r1 := WORD_TO_REAL(Rx_IH_MOUT);
pv_IH_KW := r1 / 10; 

is_IH_TIC_al := Rx_IH_AL > 0;
is_IH_TIC_manual := Rx_IH_AM > 0;
ing_IH_TIC_at := Rx_IH_AT_ST <> 0;

r1 := WORD_TO_REAL(Rx_IH_P);
pv_IH_P := r1 / 10; 

r1 := WORD_TO_REAL(Rx_IH_I);
pv_IH_I := r1 / 10; 

r1 := WORD_TO_REAL(Rx_IH_D);
pv_IH_D := r1 / 10;

END_PROGRAM

// ---- POUs/MR_PRG/P13_DI_N_Check.TcPOU
PROGRAM P13_DI_N_Check
VAR	
    T_Rst_off: TON := (PT:=T#1S);
	
	//for ACT_ROT_JOG_INCH();
	t_ROT_INCH: TON;
	pt_ROT_INCH: TIME;
	p_ROT_INCH: R_TRIG;
	p_ROT_JOG_OFF: F_TRIG;
	
	//for Maint
	p_MAINT: R_TRIG;
	p_DO_TEST: R_TRIG;
END_VAR

//for PC Display
BITS1_DI := %IB0;
BITS2_DI := %IB1;
BITS3_DI := %IB2;
BITS4_DI := %IB3;
BITS5_DI := %IB4;
BITS6_DI := %IB5;
BITS7_DI := %IB6;
BITS8_DI := %IB7;
BITS9_DI := %IB8;

//전체 Reset 신호 1초 발생
T_Rst_Off(IN:= cm_RST);
IF T_Rst_Off.Q THEN
	cm_RST := 0; 
END_IF
s_cm_RST := cm_RST;

//Maint Mode Check
p_MAINT(CLK:=(di_MAINT OR cm_MAINT));
IF p_MAINT.Q AND (di_MAINT OR cm_MAINT) AND ing_RCP = 0 AND is_MAKER_login THEN //Maint On
	ing_MAINT := 1; 
END_IF 
IF (di_MAINT = 0 AND cm_MAINT = 0) OR ing_RCP = 1 OR is_MAKER_login = 0 THEN //Maint Off
	ing_MAINT := 0; 
END_IF 

//DO Test Check
p_DO_TEST(CLK:=cm_DO_TEST);	
IF p_DO_TEST.Q AND ing_MAINT THEN
	s_EN_DO_TEST := 1; 
END_IF
IF ing_MAINT = 0 OR cm_DO_TEST = 0 THEN
	s_EN_DO_TEST := 0; 
	cm_DO_TEST := 0;
END_IF
ing_DO_TEST := s_EN_DO_TEST;	

//S01 -N2 Low Check
is_S01_low_al := pv_S01 < N_A_SV_AL[0];
is_S01_low_wn := pv_S01 < N_A_SV_WN[0];

//S02 -H2 Low Check
is_S02_low_al := pv_S02 < N_A_SV_AL[1];
is_S02_low_wn := pv_S02 < N_A_SV_WN[1];

//S03 -NH3 Low Check
is_S03_low_al := pv_S03 < N_A_SV_AL[2];
is_S03_low_wn := pv_S03 < N_A_SV_WN[2];

//S04 -SiH4 Low Check
is_S04_low_al := pv_S04 < N_A_SV_AL[3];
is_S04_low_wn := pv_S04 < N_A_SV_WN[3];

//P01 Reactor Pressure
is_P01_overP_al := pv_P01 > N_A_SV_AL[4];
is_P01_overP_wn := pv_P01 > N_A_SV_WN[4];

//IH Over Temp
is_IH_overT_al := pv_IH > N_A_SV_AL[5];
is_IH_overT_wn := pv_IH > N_A_SV_WN[5];

//Shower Head CW Over Temp
is_SH_CW_overT_al := pv_IH > N_A_SV_AL[6];
is_SH_CW_overT_wn := pv_IH > N_A_SV_WN[6];

//IH Coil CW Over Temp
is_IH_CW_overT_al := pv_IH_CW > N_A_SV_AL[7];
is_IH_CW_overT_wn := pv_IH_CW > N_A_SV_WN[7];

//P03 Exhaust Pressure
is_P03_overP_al := pv_P03 > N_A_SV_AL[8];
is_P03_overP_wn := pv_P03 > N_A_SV_WN[8];

//DOR Pressure
is_DOR_1ATM := pv_S05 >= e_DOR_1ATM;
is_DOR_05ATM := pv_S05 <= e_DOR_05ATM;
is_DOR_01ATM := pv_S05 <= e_DOR_01ATM;

is_SH_opend := di_SH_lo_limit = 0;

//Rotation : Jog & Inching
ACT_ROT_JOG_INCH();

ACTION ACT_ROT_JOG_INCH:

(*

p_ROT_JOG_OFF(CLK:=EN_ROT_JOG);
//jog runable check
EN_ROT_JOG := (di_ROT_Jog OR cm_ROT_JOG) 
				AND EN_ROT_INCH = 0 
				AND (ing_RCP = 0 OR is_ROT_caliOn = 0)  
				AND al_ROT_fail = Off;//jog
//jog speed set				
IF EN_ROT_JOG THEN
	tsv_ROT := s_ROT_JOG_SPD;
	rtm_ROT := 0;
END_IF

IF p_ROT_JOG_OFF.Q THEN
	tsv_ROT := 0;
	rtm_ROT := 0;
END_IF

t_ROT_INCH(PT := pt_ROT_INCH);//inching timer				
//inching runable check				
p_ROT_INCH(CLK := (di_ROT_60 OR cm_ROT_INCH ) AND EN_ROT_JOG = 0 AND (ing_RCP = 0 OR is_ROT_caliOn = 0) );
IF p_ROT_INCH.Q AND do_Rot = 0  THEN
	cm_ROT_INCH := Off;	
	EN_ROT_INCH := On;
END_IF

//inching speed set
IF EN_ROT_INCH THEN
	tsv_ROT := s_ROT_INCH_SPD;
	rtm_ROT := 0;
	pt_ROT_INCH := REAL_TO_TIME(s_ROT_INCH_TM);//inching time set
	t_ROT_INCH.IN := On;
END_IF

//inching end
IF t_ROT_INCH.Q OR al_ROT_fail THEN
	t_ROT_INCH.IN := Off;
	EN_ROT_INCH := Off;
	tsv_ROT := 0;
	rtm_ROT := 0;
END_IF

IF cm_ROT_pulseZero THEN
	cm_ROT_pulseZero := Off;
	pv_ROT_inchPulse := 0;
	pv_ROT_1turnPulse := 0;
END_IF

ing_ROT_jog := EN_ROT_JOG AND do_Rot;
ing_ROT_inch := EN_ROT_INCH AND do_Rot; 

*)
END_ACTION

END_PROGRAM

// ---- POUs/MR_PRG/P15_AI.TcPOU
PROGRAM P15_AI
VAR
	T1: TON := (PT:=T#100MS);
	halfRes: REAL := 16383;//0~5V
	fullRes: REAL := 32767;//0~10V or 4~20mA
	fullRes_KL3152: REAL := 65535;//4~20mA
	dorOffset: REAL := 3276;
	dorResolution: REAL := 13107;
	dorATM: REAL := 760;			
END_VAR


T1(IN:= 1);
IF T1.Q THEN
	T1(IN:= 0);
	//---------------------- ANALOG ---------------------------	
	IF N_MAX[0] > 0 THEN//MFC01 : 0~5V
	 	pv_M01 := N_MAX[0] * XA_M01 / halfRes ;
	 	dev_M01 := (100 * (sv_M01 - pv_M01)) / N_MAX[0];
	END_IF;	
	IF N_MAX[1] > 0 THEN//MFC02 : 0~5V
		pv_M02 := N_MAX[1] * XA_M02 / halfRes ;
	 	dev_M02 := (100 * (sv_M02 - pv_M02)) / N_MAX[1];
	END_IF;	
	IF N_MAX[2] > 0 THEN//MFC03 : 0~5V
		 pv_M03 := N_MAX[2] * XA_M03 / halfRes ;
		 dev_M03 := (100 * (sv_M03 - pv_M03)) / N_MAX[2];
	END_IF;	
	IF N_MAX[3] > 0 THEN//MFC04 : 0~5V
		 pv_M04 := N_MAX[3] * XA_M04 / halfRes ;
		 dev_M04 := (100 * (sv_M04 - pv_M04)) / N_MAX[3];
	END_IF;	
	IF N_MAX[4] > 0 THEN//MFC05 : 0~5V
		 pv_M05 := N_MAX[4] * XA_M05 / halfRes ;
		 dev_M05 := (100 * (sv_M05 - pv_M05)) / N_MAX[4];
	END_IF;	
	IF N_MAX[5] > 0 THEN//MFC06 : 0~5V
		 pv_M06 := N_MAX[5] * XA_M06 / halfRes ;
		 dev_M06 := (100 * (sv_M06 - pv_M06)) / N_MAX[5];
	END_IF;	
	IF N_MAX[6] > 0 THEN//MFC07 : 0~5V
		 pv_M07 := N_MAX[6] * XA_M07 / halfRes ;
		 dev_M07 := (100 * (sv_M07 - pv_M07)) / N_MAX[6];
	END_IF;	
	IF N_MAX[7] > 0 THEN//MFC08 : 0~5V
		 pv_M08 := N_MAX[7] * XA_M08 / halfRes ;
		 dev_M08 := (100 * (sv_M08 - pv_M08)) / N_MAX[7];
	END_IF;	
	IF N_MAX[8] > 0 THEN//MFC09 : 0~5V
		 pv_M09 := N_MAX[8] * XA_M09 / halfRes ;
		 dev_M09 := (100 * (sv_M09 - pv_M09)) / N_MAX[8];
	END_IF;	
	IF N_MAX[9] > 0 THEN//MFC10 : 0~5V
		 pv_M10 := N_MAX[9] * XA_M10 / halfRes ;
		 dev_M10 := (100 * (sv_M10 - pv_M10)) / N_MAX[9];
	END_IF;	
	IF N_MAX[10] > 0 THEN//MFC11 : 0~5V
		 pv_M11 := N_MAX[10] * XA_M11 / halfRes ;
		 dev_M11 := (100 * (sv_M11 - pv_M11)) / N_MAX[10];
	END_IF;	
	IF N_MAX[11] > 0 THEN//MFC12 : 0~5V
		 pv_M12 := N_MAX[11] * XA_M12 / halfRes ;
		 dev_M12 := (100 * (sv_M12 - pv_M12)) / N_MAX[11];
	END_IF;	
	IF N_MAX[12] > 0 THEN//MFC13 : 0~5V
		 pv_M13 := N_MAX[12] * XA_M13 / halfRes ;
		 dev_M13 := (100 * (sv_M13 - pv_M13)) / N_MAX[12];
	END_IF;	
	IF N_MAX[13] > 0 THEN//MFC14 : 0~5V
		 pv_M14 := N_MAX[13] * XA_M14 / halfRes ;
		 dev_M14 := (100 * (sv_M14 - pv_M14)) / N_MAX[13];
	END_IF;	
	IF N_MAX[14] > 0 THEN//MFC15 : 0~5V
		 pv_M15 := N_MAX[14] * XA_M15 / halfRes ;
		 dev_M15 := (100 * (sv_M15 - pv_M15)) / N_MAX[14];
	END_IF;	
	IF N_MAX[15] > 0 THEN//MFC16 : 0~5V
	 	pv_M16 := N_MAX[15] * XA_M16 / halfRes ;
	 	dev_M16 := (100 * (sv_M16 - pv_M16)) / N_MAX[15];
	END_IF;	
	IF N_MAX[16] > 0 THEN//MFC17 : 0~5V
		 pv_M17 := N_MAX[16] * XA_M17 / halfRes ;
		 dev_M17 := (100 * (sv_M17 - pv_M17)) / N_MAX[16];
	END_IF;	
	IF N_MAX[17] > 0 THEN//MFC18 : 0~5V
		 pv_M18 := N_MAX[17] * XA_M18 / halfRes ;
		 dev_M18 := (100 * (sv_M18 - pv_M18)) / N_MAX[17];
	END_IF;	
	IF N_MAX[18] > 0 THEN//MFC19 : 0~5V
		 pv_M19 := N_MAX[18] * XA_M19 / halfRes ;
		 dev_M19 := (100 * (sv_M19 - pv_M19)) / N_MAX[18];
	END_IF;				
	IF N_MAX[19] > 0 THEN//EPC01 : 0~5V
		pv_E01 := N_MAX[19] * XA_E01 / halfRes ;
		dev_E01 := (100 * (sv_E01 - pv_E01)) / N_MAX[19];
	END_IF;	
	IF N_MAX[20] > 0 THEN//EPC02 : 0~5V
		pv_E02 := N_MAX[20] * XA_E02 / halfRes ;
		dev_E02 := (100 * (sv_E02 - pv_E02)) / N_MAX[20];
	END_IF;	
	IF N_MAX[21] > 0 THEN//EPC03 : 0~5V
		pv_E03 := N_MAX[21] * XA_E03 / halfRes ;
		dev_E03 := (100 * (sv_E03 - pv_E03)) / N_MAX[21];
	END_IF;	
	IF N_MAX[22] > 0 THEN//EPC04 : 0~5V
		pv_E04 := N_MAX[22] * XA_E04 / halfRes ;
		dev_E04 := (100 * (sv_E04 - pv_E04)) / N_MAX[22];
	END_IF;	
	IF N_MAX[23] > 0 THEN //EPC05 : 0~5V
		pv_E05 := N_MAX[23] * XA_E05 / halfRes ;
		dev_E05 := (100 * (sv_E05 - pv_E05)) / N_MAX[23];
	END_IF;	
	IF N_MAX[24] > 0 THEN //EPC06 : 0~5V
		pv_E06 := N_MAX[24] * XA_E06 / halfRes ;
		dev_E06 := (100 * (sv_E06 - pv_E06)) / N_MAX[24];
	END_IF;
	IF N_MAX[25] > 0 THEN//EPC07 : 0~5V
		pv_E07 := N_MAX[25] * XA_E07 / halfRes ;
		dev_E07 := (100 * (sv_E07 - pv_E07)) / N_MAX[25];
	END_IF;			
	IF N_MAX[26] > 0 THEN//IH Temp - E3508 
		//pv_IHT := DeviceNet
		dev_IH := (100 * (sv_IH - pv_IH)) / N_MAX[26];
	END_IF;	
	IF N_MAX[27] > 0 THEN//Rotation RPM : 4~20mA      
	   	 pv_Rot := N_MAX[27] * XA_ROT / fullRes_KL3152;
		 dev_ROT := (100 * (sv_ROT - pv_ROT)) / N_MAX[27];
	END_IF;	
	IF N_MAX[28] > 0 THEN//T/V Position(1~100%) : DeviceNet
		//pv_TV := DeviceNet
		dev_POS := (100 * (sv_POS - pv_POS)) / N_MAX[28];
	END_IF;
	IF N_MAX[29] > 0 THEN//T/V Pressure(1~1000 Torr) : DeviceNet
		//pv_P01 := DeviceNet
		dev_P01 := (100 * (sv_P01 - pv_P01)) / N_MAX[29];
	END_IF;	
	IF N_MAX[30] > 0 THEN//Reactor Pressure(10 Torr) : 0~10V
		pv_P02 := N_MAX[30] * XA_P02 / fullRes;
	END_IF;	
	IF N_MAX[31] > 0 THEN//Exhaust Pressure(1000 Torr) : 0~10V   
	   	 pv_P03 := N_MAX[31] * XA_P03 / fullRes;
	END_IF;		
	IF N_MAX[52] > 0 THEN//N2 Pressure : 4~20mA      
		 pv_S01 := N_MAX[52] * XA_S01 / fullRes;
	END_IF;	
	IF N_MAX[53] > 0 THEN//H2 Pressure : 4~20mA      
		 pv_S02 := N_MAX[53] * XA_S02 / fullRes;
	END_IF;	
	IF N_MAX[54] > 0 THEN//NH3 Pressure : 4~20mA       
		 pv_S03 := N_MAX[54] * XA_S03 / fullRes;
	END_IF;	 
	IF N_MAX[55] > 0 THEN//SiH4 Pressure : 4~20mA      
		 pv_S04 := N_MAX[55] * XA_S04 / fullRes;
	END_IF;	
	IF N_MAX[56] > 0 THEN//DOR Pressure : 1~5V      
		 pv_S05 :=  dorATM - (N_MAX[56] * (XA_S05 - dorOffset) / dorResolution);
	END_IF;
				
	//pv_LHT1 := XA_LHT1 * 0.1 ;
	//pv_LHT2 := XA_LHT2 * 0.1 ;
	//pv_LHT3 := XA_LHT3 * 0.1 ;
	//pv_LHT4 := XA_LHT4 * 0.1 ;
	//pv_LHT5 := XA_LHT5 * 0.1 ;
	//pv_LHT6 := XA_LHT6 * 0.1 ;
	//pv_LHT7 := XA_LHT7 * 0.1 ;
	//pv_LHT8 := XA_LHT8 * 0.1 ;
		
	//Shower Head Temp.
	pv_SH_CW  := XA_SH_CW * 0.1 ;	
	//Induction Coil Water Temp
	pv_IH_CW := XA_IH_CW * 0.1 ;
		
    //Induction KW

END_IF;

END_PROGRAM

// ---- POUs/MR_PRG/P21_AL_WN.TcPOU
PROGRAM P21_AL_WN
VAR
	//Analog Deviation Check
	Dev00, Dev01, Dev02, Dev03, Dev04, Dev05, Dev06, Dev07, Dev08, Dev09: FB_DeviationCheck;
	Dev10, Dev11, Dev12, Dev13, Dev14, Dev15, Dev16, Dev17, Dev18, Dev19: FB_DeviationCheck;
	Dev20, Dev21, Dev22, Dev23, Dev24, Dev25, Dev26, Dev27, Dev28, Dev29: FB_DeviationCheck;
		
	//Digital Noise Check
	wNoiseCheckTime: WORD := 100;	
	FB_AL32, FB_AL33, FB_AL34, FB_AL35, FB_AL36, FB_AL37, FB_AL38, FB_AL39: FB_NoiseCheck;	 
	FB_AL40, FB_AL41, FB_AL42, FB_AL43, FB_AL44, FB_AL45, FB_AL46, FB_AL47: FB_NoiseCheck;
	FB_AL48, FB_AL49, FB_AL50, FB_AL51, FB_AL52, FB_AL53, FB_AL54, FB_AL55: FB_NoiseCheck; 
	FB_AL56, FB_AL57, FB_AL58, FB_AL59, FB_AL60, FB_AL61, FB_AL62, FB_AL63: FB_NoiseCheck; 
	FB_AL64, FB_AL65, FB_AL66, FB_AL67, FB_AL68, FB_AL69, FB_AL70, FB_AL71: FB_NoiseCheck; 
	FB_AL72, FB_AL73, FB_AL74, FB_AL75, FB_AL76, FB_AL77, FB_AL78, FB_AL79: FB_NoiseCheck; 
	FB_AL80, FB_AL81, FB_AL82, FB_AL83, FB_AL84, FB_AL85, FB_AL86, FB_AL87: FB_NoiseCheck;
	FB_AL88, FB_AL89, FB_AL90, FB_AL91, FB_AL92, FB_AL93, FB_AL94, FB_AL95: FB_NoiseCheck; 
	FB_AL96, FB_AL97, FB_AL98, FB_AL99, FB_AL100, FB_AL101, FB_AL102, FB_AL103: FB_NoiseCheck; 
	FB_AL104, FB_AL105, FB_AL106, FB_AL107, FB_AL108, FB_AL109, FB_AL110, FB_AL111: FB_NoiseCheck;
	//FB_AL112, FB_AL113, FB_AL114, FB_AL115, FB_AL116, FB_AL117, FB_AL118, FB_AL119: FB_NoiseCheck; 
	FB_AL120, FB_AL121, FB_AL122, FB_AL123, FB_AL124, FB_AL125, FB_AL126, FB_AL127: FB_NoiseCheck;
	FB_AL128, FB_AL129, FB_AL130, FB_AL131, FB_AL132, FB_AL133, FB_AL134, FB_AL135: FB_NoiseCheck;
	FB_AL136, FB_AL137, FB_AL138, FB_AL139, FB_AL140, FB_AL141, FB_AL142, FB_AL143: FB_NoiseCheck;
	//FB_AL144, FB_AL145, FB_AL146, FB_AL147, FB_AL148, FB_AL149, FB_AL150, FB_AL151: FB_NoiseCheck;
	//FB_AL152, FB_AL153, FB_AL154, FB_AL155, FB_AL156, FB_AL157, FB_AL158, FB_AL159: FB_NoiseCheck;	
			
	FB_WN32, FB_WN33, FB_WN34, FB_WN35, FB_WN36, FB_WN37, FB_WN38, FB_WN39: FB_NoiseCheck; 
	FB_WN40, FB_WN41, FB_WN42, FB_WN43, FB_WN44, FB_WN45, FB_WN46, FB_WN47, FB_WN48, FB_WN49: FB_NoiseCheck; 
	FB_WN50, FB_WN51, FB_WN52, FB_WN53, FB_WN54, FB_WN55, FB_WN56, FB_WN57, FB_WN58, FB_WN59: FB_NoiseCheck; 
	FB_WN60, FB_WN61, FB_WN62, FB_WN63: FB_NoiseCheck;
									
	i: INT;
	bReset: BOOL;
	P_AL_Trig: R_TRIG;
	P_WN_Trig: R_TRIG;
	
	P_di_RST: R_TRIG;
		
	//Real Address
	n_AL_WORD AT%MB38: ARRAY[0..8] OF WORD; //16Bit
	n_WN_DWORD AT%MB56: ARRAY[0..1] OF DWORD; //32Bit
		
	n_AL_WORD_OLD: ARRAY[0..8] OF DWORD; //128EA
	n_WN_DWORD_OLD: ARRAY[0..1] OF DWORD; //64EA
	
	T1S_WN: TON;
	n_BZ_Order: ARRAY[0..1] OF BYTE;//부저 울림 순서, 1 -> Warning, 2 -> Alarm, 1 + 2 = 3 -> Alarm

END_VAR

A_AL_WN_Check();
D_AL_Check();
D_WN_Check();

is_AL := n_AL_WORD[0] > 0 OR n_AL_WORD[1] > 0 OR n_AL_WORD[2] > 0 OR n_AL_WORD[3] > 0 OR n_AL_WORD[4] > 0 OR
		 n_AL_WORD[5] > 0 OR n_AL_WORD[6] > 0 OR n_AL_WORD[7] > 0 OR n_AL_WORD[8] > 0;

is_WN := n_WN_DWORD[0] > 0 OR n_WN_DWORD[1] > 0 ;

//Alarm Processing
D_AL_Check();

//Alarm & Warning Reset
bReset := s_cm_RST;
 IF bReset THEN
	 s_is_DOR_Broken := 0;
 END_IF

//New AL Check
P_AL_Trig(CLK:= n_AL_WORD[0] > n_AL_WORD_OLD[0] OR n_AL_WORD[1] > n_AL_WORD_OLD[1] OR 
			  n_AL_WORD[2] > n_AL_WORD_OLD[2] OR n_AL_WORD[3] > n_AL_WORD_OLD[3] OR
			  n_AL_WORD[4] > n_AL_WORD_OLD[4] OR n_AL_WORD[5] > n_AL_WORD_OLD[5] OR
			  n_AL_WORD[6] > n_AL_WORD_OLD[6] OR n_AL_WORD[7] > n_AL_WORD_OLD[7] OR
			  n_AL_WORD[8] > n_AL_WORD_OLD[8]);
//New WN Check	
P_WN_Trig(CLK:= n_WN_DWORD[0] > n_WN_DWORD_OLD[0] OR n_WN_DWORD[1] > n_WN_DWORD_OLD[1]);

P_di_RST(CLK:= di_RST);	

//AL Backup	
FOR i := 0 TO 8 DO
	n_AL_WORD_OLD[i] := n_AL_WORD[i];
END_FOR
//WN Backup
FOR i := 0 TO 1 DO
	n_WN_DWORD_OLD[i] := n_WN_DWORD[i];
END_FOR

ACTION A_AL_WN_Check:
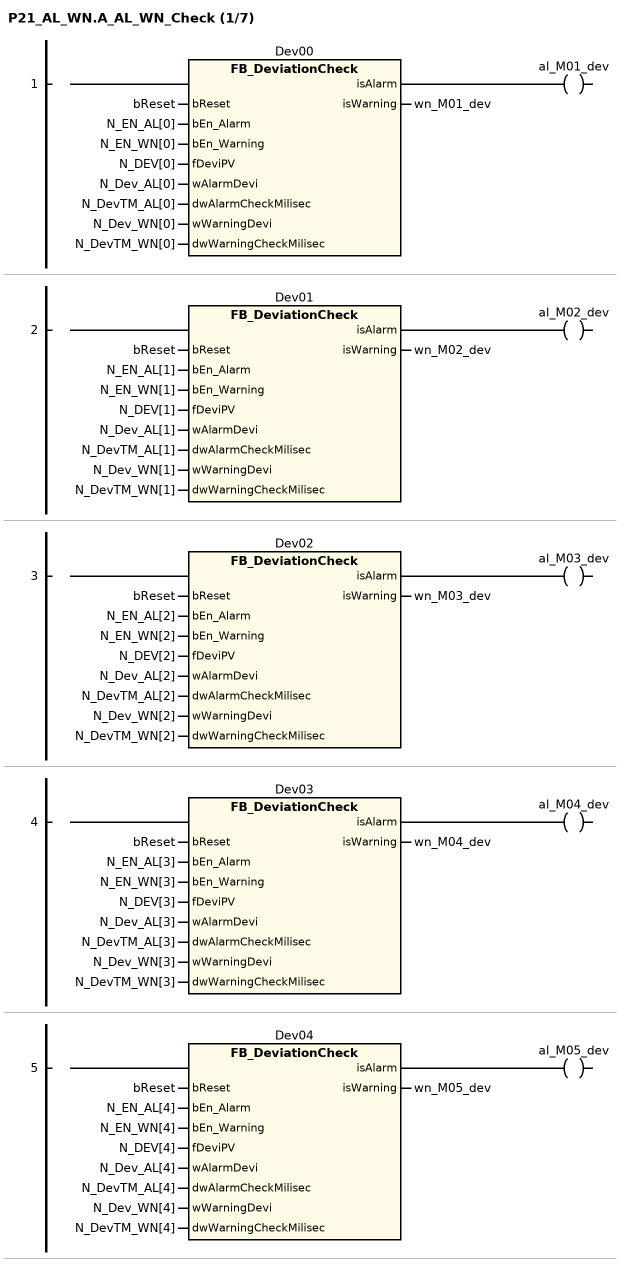
// NETWORK 1
Dev00(
    bReset := bReset,
    bEn_Alarm := N_EN_AL[0],
    bEn_Warning := N_EN_WN[0],
    fDeviPV := N_DEV[0],
    wAlarmDevi := N_Dev_AL[0],
    dwAlarmCheckMilisec := N_DevTM_AL[0],
    wWarningDevi := N_Dev_WN[0],
    dwWarningCheckMilisec := N_DevTM_WN[0],
    isWarning => wn_M01_dev); // FB_DeviationCheck
al_M01_dev := Dev00.isAlarm;

// NETWORK 2
Dev01(
    bReset := bReset,
    bEn_Alarm := N_EN_AL[1],
    bEn_Warning := N_EN_WN[1],
    fDeviPV := N_DEV[1],
    wAlarmDevi := N_Dev_AL[1],
    dwAlarmCheckMilisec := N_DevTM_AL[1],
    wWarningDevi := N_Dev_WN[1],
    dwWarningCheckMilisec := N_DevTM_WN[1],
    isWarning => wn_M02_dev); // FB_DeviationCheck
al_M02_dev := Dev01.isAlarm;

// NETWORK 3
Dev02(
    bReset := bReset,
    bEn_Alarm := N_EN_AL[2],
    bEn_Warning := N_EN_WN[2],
    fDeviPV := N_DEV[2],
    wAlarmDevi := N_Dev_AL[2],
    dwAlarmCheckMilisec := N_DevTM_AL[2],
    wWarningDevi := N_Dev_WN[2],
    dwWarningCheckMilisec := N_DevTM_WN[2],
    isWarning => wn_M03_dev); // FB_DeviationCheck
al_M03_dev := Dev02.isAlarm;

// NETWORK 4
Dev03(
    bReset := bReset,
    bEn_Alarm := N_EN_AL[3],
    bEn_Warning := N_EN_WN[3],
    fDeviPV := N_DEV[3],
    wAlarmDevi := N_Dev_AL[3],
    dwAlarmCheckMilisec := N_DevTM_AL[3],
    wWarningDevi := N_Dev_WN[3],
    dwWarningCheckMilisec := N_DevTM_WN[3],
    isWarning => wn_M04_dev); // FB_DeviationCheck
al_M04_dev := Dev03.isAlarm;

// NETWORK 5
Dev04(
    bReset := bReset,
    bEn_Alarm := N_EN_AL[4],
    bEn_Warning := N_EN_WN[4],
    fDeviPV := N_DEV[4],
    wAlarmDevi := N_Dev_AL[4],
    dwAlarmCheckMilisec := N_DevTM_AL[4],
    wWarningDevi := N_Dev_WN[4],
    dwWarningCheckMilisec := N_DevTM_WN[4],
    isWarning => wn_M05_dev); // FB_DeviationCheck
al_M05_dev := Dev04.isAlarm;

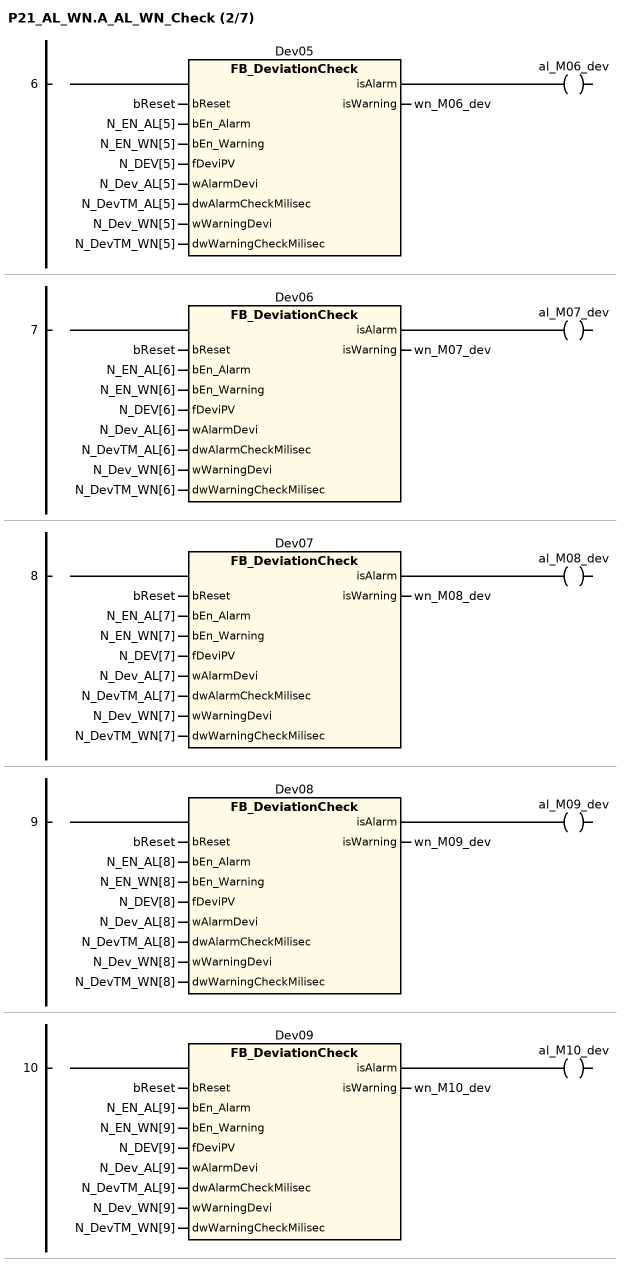
// NETWORK 6
Dev05(
    bReset := bReset,
    bEn_Alarm := N_EN_AL[5],
    bEn_Warning := N_EN_WN[5],
    fDeviPV := N_DEV[5],
    wAlarmDevi := N_Dev_AL[5],
    dwAlarmCheckMilisec := N_DevTM_AL[5],
    wWarningDevi := N_Dev_WN[5],
    dwWarningCheckMilisec := N_DevTM_WN[5],
    isWarning => wn_M06_dev); // FB_DeviationCheck
al_M06_dev := Dev05.isAlarm;

// NETWORK 7
Dev06(
    bReset := bReset,
    bEn_Alarm := N_EN_AL[6],
    bEn_Warning := N_EN_WN[6],
    fDeviPV := N_DEV[6],
    wAlarmDevi := N_Dev_AL[6],
    dwAlarmCheckMilisec := N_DevTM_AL[6],
    wWarningDevi := N_Dev_WN[6],
    dwWarningCheckMilisec := N_DevTM_WN[6],
    isWarning => wn_M07_dev); // FB_DeviationCheck
al_M07_dev := Dev06.isAlarm;

// NETWORK 8
Dev07(
    bReset := bReset,
    bEn_Alarm := N_EN_AL[7],
    bEn_Warning := N_EN_WN[7],
    fDeviPV := N_DEV[7],
    wAlarmDevi := N_Dev_AL[7],
    dwAlarmCheckMilisec := N_DevTM_AL[7],
    wWarningDevi := N_Dev_WN[7],
    dwWarningCheckMilisec := N_DevTM_WN[7],
    isWarning => wn_M08_dev); // FB_DeviationCheck
al_M08_dev := Dev07.isAlarm;

// NETWORK 9
Dev08(
    bReset := bReset,
    bEn_Alarm := N_EN_AL[8],
    bEn_Warning := N_EN_WN[8],
    fDeviPV := N_DEV[8],
    wAlarmDevi := N_Dev_AL[8],
    dwAlarmCheckMilisec := N_DevTM_AL[8],
    wWarningDevi := N_Dev_WN[8],
    dwWarningCheckMilisec := N_DevTM_WN[8],
    isWarning => wn_M09_dev); // FB_DeviationCheck
al_M09_dev := Dev08.isAlarm;

// NETWORK 10
Dev09(
    bReset := bReset,
    bEn_Alarm := N_EN_AL[9],
    bEn_Warning := N_EN_WN[9],
    fDeviPV := N_DEV[9],
    wAlarmDevi := N_Dev_AL[9],
    dwAlarmCheckMilisec := N_DevTM_AL[9],
    wWarningDevi := N_Dev_WN[9],
    dwWarningCheckMilisec := N_DevTM_WN[9],
    isWarning => wn_M10_dev); // FB_DeviationCheck
al_M10_dev := Dev09.isAlarm;

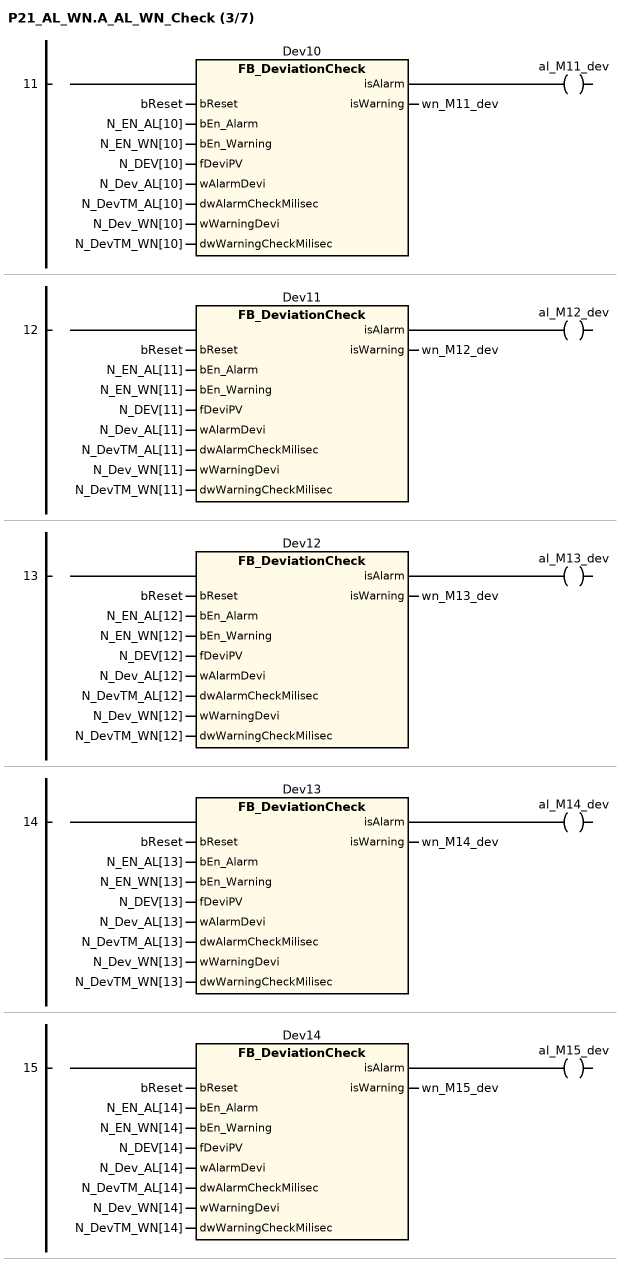
// NETWORK 11
Dev10(
    bReset := bReset,
    bEn_Alarm := N_EN_AL[10],
    bEn_Warning := N_EN_WN[10],
    fDeviPV := N_DEV[10],
    wAlarmDevi := N_Dev_AL[10],
    dwAlarmCheckMilisec := N_DevTM_AL[10],
    wWarningDevi := N_Dev_WN[10],
    dwWarningCheckMilisec := N_DevTM_WN[10],
    isWarning => wn_M11_dev); // FB_DeviationCheck
al_M11_dev := Dev10.isAlarm;

// NETWORK 12
Dev11(
    bReset := bReset,
    bEn_Alarm := N_EN_AL[11],
    bEn_Warning := N_EN_WN[11],
    fDeviPV := N_DEV[11],
    wAlarmDevi := N_Dev_AL[11],
    dwAlarmCheckMilisec := N_DevTM_AL[11],
    wWarningDevi := N_Dev_WN[11],
    dwWarningCheckMilisec := N_DevTM_WN[11],
    isWarning => wn_M12_dev); // FB_DeviationCheck
al_M12_dev := Dev11.isAlarm;

// NETWORK 13
Dev12(
    bReset := bReset,
    bEn_Alarm := N_EN_AL[12],
    bEn_Warning := N_EN_WN[12],
    fDeviPV := N_DEV[12],
    wAlarmDevi := N_Dev_AL[12],
    dwAlarmCheckMilisec := N_DevTM_AL[12],
    wWarningDevi := N_Dev_WN[12],
    dwWarningCheckMilisec := N_DevTM_WN[12],
    isWarning => wn_M13_dev); // FB_DeviationCheck
al_M13_dev := Dev12.isAlarm;

// NETWORK 14
Dev13(
    bReset := bReset,
    bEn_Alarm := N_EN_AL[13],
    bEn_Warning := N_EN_WN[13],
    fDeviPV := N_DEV[13],
    wAlarmDevi := N_Dev_AL[13],
    dwAlarmCheckMilisec := N_DevTM_AL[13],
    wWarningDevi := N_Dev_WN[13],
    dwWarningCheckMilisec := N_DevTM_WN[13],
    isWarning => wn_M14_dev); // FB_DeviationCheck
al_M14_dev := Dev13.isAlarm;

// NETWORK 15
Dev14(
    bReset := bReset,
    bEn_Alarm := N_EN_AL[14],
    bEn_Warning := N_EN_WN[14],
    fDeviPV := N_DEV[14],
    wAlarmDevi := N_Dev_AL[14],
    dwAlarmCheckMilisec := N_DevTM_AL[14],
    wWarningDevi := N_Dev_WN[14],
    dwWarningCheckMilisec := N_DevTM_WN[14],
    isWarning => wn_M15_dev); // FB_DeviationCheck
al_M15_dev := Dev14.isAlarm;

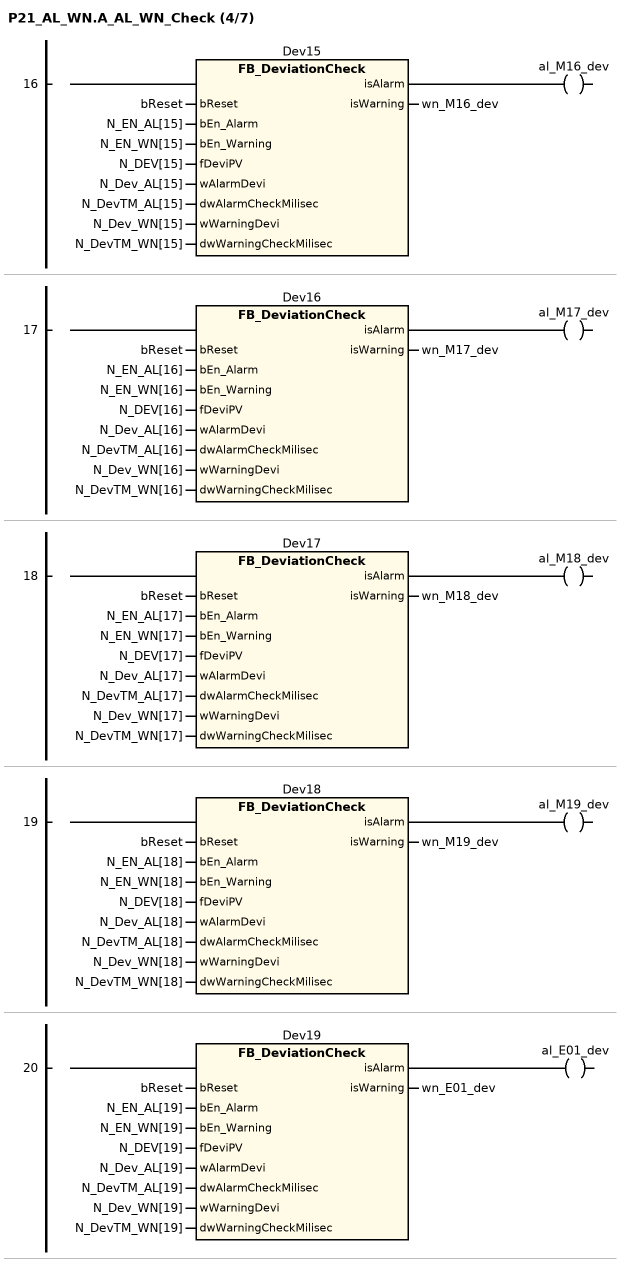
// NETWORK 16
Dev15(
    bReset := bReset,
    bEn_Alarm := N_EN_AL[15],
    bEn_Warning := N_EN_WN[15],
    fDeviPV := N_DEV[15],
    wAlarmDevi := N_Dev_AL[15],
    dwAlarmCheckMilisec := N_DevTM_AL[15],
    wWarningDevi := N_Dev_WN[15],
    dwWarningCheckMilisec := N_DevTM_WN[15],
    isWarning => wn_M16_dev); // FB_DeviationCheck
al_M16_dev := Dev15.isAlarm;

// NETWORK 17
Dev16(
    bReset := bReset,
    bEn_Alarm := N_EN_AL[16],
    bEn_Warning := N_EN_WN[16],
    fDeviPV := N_DEV[16],
    wAlarmDevi := N_Dev_AL[16],
    dwAlarmCheckMilisec := N_DevTM_AL[16],
    wWarningDevi := N_Dev_WN[16],
    dwWarningCheckMilisec := N_DevTM_WN[16],
    isWarning => wn_M17_dev); // FB_DeviationCheck
al_M17_dev := Dev16.isAlarm;

// NETWORK 18
Dev17(
    bReset := bReset,
    bEn_Alarm := N_EN_AL[17],
    bEn_Warning := N_EN_WN[17],
    fDeviPV := N_DEV[17],
    wAlarmDevi := N_Dev_AL[17],
    dwAlarmCheckMilisec := N_DevTM_AL[17],
    wWarningDevi := N_Dev_WN[17],
    dwWarningCheckMilisec := N_DevTM_WN[17],
    isWarning => wn_M18_dev); // FB_DeviationCheck
al_M18_dev := Dev17.isAlarm;

// NETWORK 19
Dev18(
    bReset := bReset,
    bEn_Alarm := N_EN_AL[18],
    bEn_Warning := N_EN_WN[18],
    fDeviPV := N_DEV[18],
    wAlarmDevi := N_Dev_AL[18],
    dwAlarmCheckMilisec := N_DevTM_AL[18],
    wWarningDevi := N_Dev_WN[18],
    dwWarningCheckMilisec := N_DevTM_WN[18],
    isWarning => wn_M19_dev); // FB_DeviationCheck
al_M19_dev := Dev18.isAlarm;

// NETWORK 20
Dev19(
    bReset := bReset,
    bEn_Alarm := N_EN_AL[19],
    bEn_Warning := N_EN_WN[19],
    fDeviPV := N_DEV[19],
    wAlarmDevi := N_Dev_AL[19],
    dwAlarmCheckMilisec := N_DevTM_AL[19],
    wWarningDevi := N_Dev_WN[19],
    dwWarningCheckMilisec := N_DevTM_WN[19],
    isWarning => wn_E01_dev); // FB_DeviationCheck
al_E01_dev := Dev19.isAlarm;

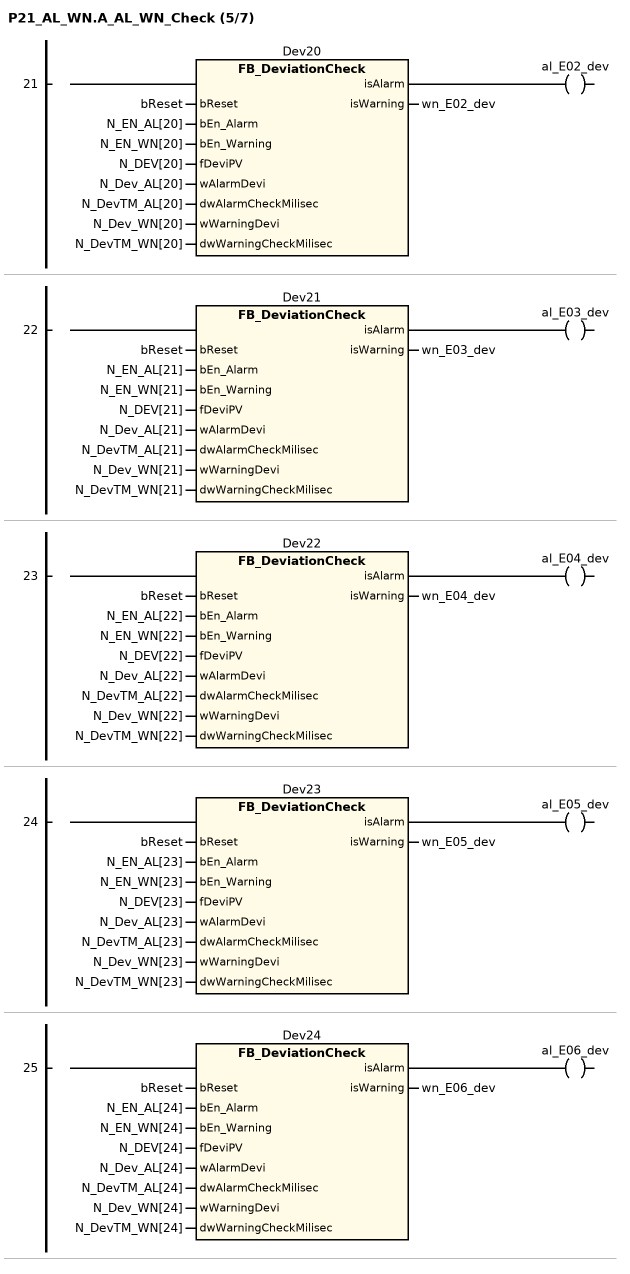
// NETWORK 21
Dev20(
    bReset := bReset,
    bEn_Alarm := N_EN_AL[20],
    bEn_Warning := N_EN_WN[20],
    fDeviPV := N_DEV[20],
    wAlarmDevi := N_Dev_AL[20],
    dwAlarmCheckMilisec := N_DevTM_AL[20],
    wWarningDevi := N_Dev_WN[20],
    dwWarningCheckMilisec := N_DevTM_WN[20],
    isWarning => wn_E02_dev); // FB_DeviationCheck
al_E02_dev := Dev20.isAlarm;

// NETWORK 22
Dev21(
    bReset := bReset,
    bEn_Alarm := N_EN_AL[21],
    bEn_Warning := N_EN_WN[21],
    fDeviPV := N_DEV[21],
    wAlarmDevi := N_Dev_AL[21],
    dwAlarmCheckMilisec := N_DevTM_AL[21],
    wWarningDevi := N_Dev_WN[21],
    dwWarningCheckMilisec := N_DevTM_WN[21],
    isWarning => wn_E03_dev); // FB_DeviationCheck
al_E03_dev := Dev21.isAlarm;

// NETWORK 23
Dev22(
    bReset := bReset,
    bEn_Alarm := N_EN_AL[22],
    bEn_Warning := N_EN_WN[22],
    fDeviPV := N_DEV[22],
    wAlarmDevi := N_Dev_AL[22],
    dwAlarmCheckMilisec := N_DevTM_AL[22],
    wWarningDevi := N_Dev_WN[22],
    dwWarningCheckMilisec := N_DevTM_WN[22],
    isWarning => wn_E04_dev); // FB_DeviationCheck
al_E04_dev := Dev22.isAlarm;

// NETWORK 24
Dev23(
    bReset := bReset,
    bEn_Alarm := N_EN_AL[23],
    bEn_Warning := N_EN_WN[23],
    fDeviPV := N_DEV[23],
    wAlarmDevi := N_Dev_AL[23],
    dwAlarmCheckMilisec := N_DevTM_AL[23],
    wWarningDevi := N_Dev_WN[23],
    dwWarningCheckMilisec := N_DevTM_WN[23],
    isWarning => wn_E05_dev); // FB_DeviationCheck
al_E05_dev := Dev23.isAlarm;

// NETWORK 25
Dev24(
    bReset := bReset,
    bEn_Alarm := N_EN_AL[24],
    bEn_Warning := N_EN_WN[24],
    fDeviPV := N_DEV[24],
    wAlarmDevi := N_Dev_AL[24],
    dwAlarmCheckMilisec := N_DevTM_AL[24],
    wWarningDevi := N_Dev_WN[24],
    dwWarningCheckMilisec := N_DevTM_WN[24],
    isWarning => wn_E06_dev); // FB_DeviationCheck
al_E06_dev := Dev24.isAlarm;

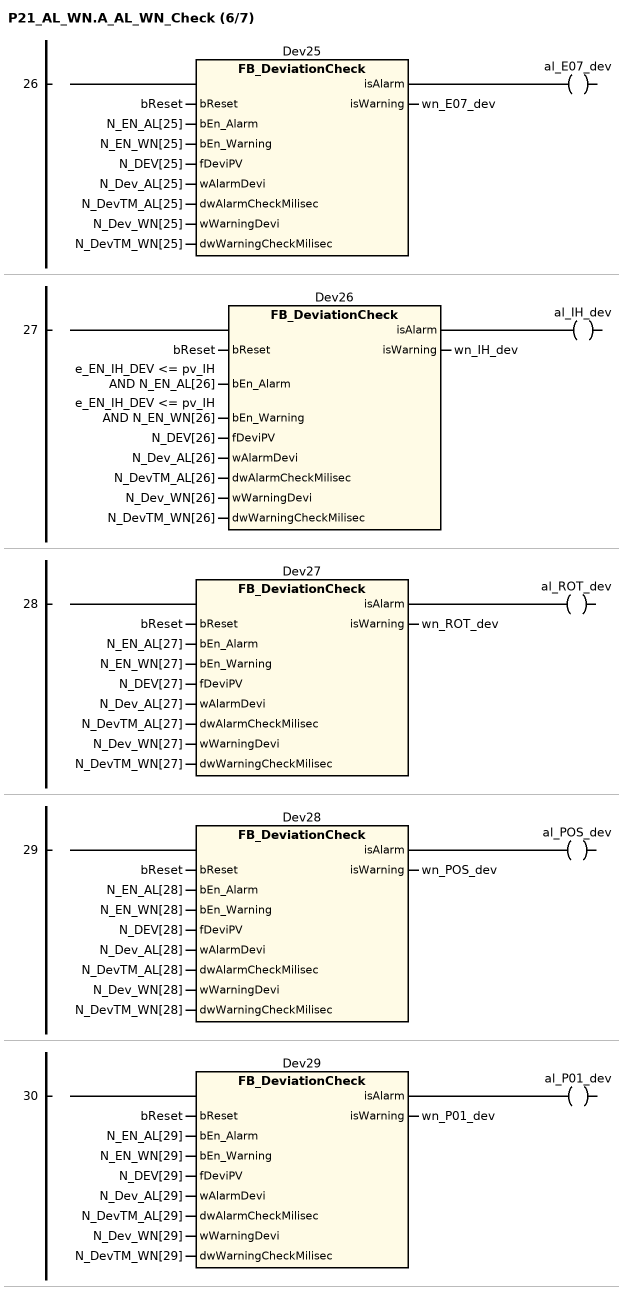
// NETWORK 26
Dev25(
    bReset := bReset,
    bEn_Alarm := N_EN_AL[25],
    bEn_Warning := N_EN_WN[25],
    fDeviPV := N_DEV[25],
    wAlarmDevi := N_Dev_AL[25],
    dwAlarmCheckMilisec := N_DevTM_AL[25],
    wWarningDevi := N_Dev_WN[25],
    dwWarningCheckMilisec := N_DevTM_WN[25],
    isWarning => wn_E07_dev); // FB_DeviationCheck
al_E07_dev := Dev25.isAlarm;

// NETWORK 27
Dev26(
    bReset := bReset,
    bEn_Alarm := e_EN_IH_DEV <= pv_IH AND N_EN_AL[26],
    bEn_Warning := e_EN_IH_DEV <= pv_IH AND N_EN_WN[26],
    fDeviPV := N_DEV[26],
    wAlarmDevi := N_Dev_AL[26],
    dwAlarmCheckMilisec := N_DevTM_AL[26],
    wWarningDevi := N_Dev_WN[26],
    dwWarningCheckMilisec := N_DevTM_WN[26],
    isWarning => wn_IH_dev); // FB_DeviationCheck
al_IH_dev := Dev26.isAlarm;

// NETWORK 28
Dev27(
    bReset := bReset,
    bEn_Alarm := N_EN_AL[27],
    bEn_Warning := N_EN_WN[27],
    fDeviPV := N_DEV[27],
    wAlarmDevi := N_Dev_AL[27],
    dwAlarmCheckMilisec := N_DevTM_AL[27],
    wWarningDevi := N_Dev_WN[27],
    dwWarningCheckMilisec := N_DevTM_WN[27],
    isWarning => wn_ROT_dev); // FB_DeviationCheck
al_ROT_dev := Dev27.isAlarm;

// NETWORK 29
Dev28(
    bReset := bReset,
    bEn_Alarm := N_EN_AL[28],
    bEn_Warning := N_EN_WN[28],
    fDeviPV := N_DEV[28],
    wAlarmDevi := N_Dev_AL[28],
    dwAlarmCheckMilisec := N_DevTM_AL[28],
    wWarningDevi := N_Dev_WN[28],
    dwWarningCheckMilisec := N_DevTM_WN[28],
    isWarning => wn_POS_dev); // FB_DeviationCheck
al_POS_dev := Dev28.isAlarm;

// NETWORK 30
Dev29(
    bReset := bReset,
    bEn_Alarm := N_EN_AL[29],
    bEn_Warning := N_EN_WN[29],
    fDeviPV := N_DEV[29],
    wAlarmDevi := N_Dev_AL[29],
    dwAlarmCheckMilisec := N_DevTM_AL[29],
    wWarningDevi := N_Dev_WN[29],
    dwWarningCheckMilisec := N_DevTM_WN[29],
    isWarning => wn_P01_dev); // FB_DeviationCheck
al_P01_dev := Dev29.isAlarm;

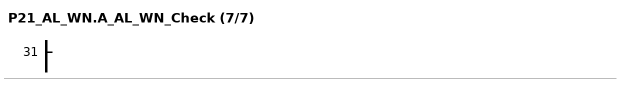
// NETWORK 31
END_ACTION

ACTION Cause_N_Effect:

//WN Buzzer
IF P_WN_Trig.Q THEN
	IF n_BZ_Order[0] <= 0 THEN
		n_BZ_Order[0] := 1; 
	ELSE
		IF n_BZ_Order[0] <> 1 THEN
			n_BZ_Order[1] := 1;
		END_IF
	END_IF
END_IF

//new Alarm rised
IF P_AL_Trig.Q THEN	
	//AL Buzzer
	IF n_BZ_Order[0] <= 0 THEN
		n_BZ_Order[0] := 2; 
	ELSE
		IF n_BZ_Order[0] <> 2 THEN
			n_BZ_Order[1] := 2;
		END_IF
	END_IF
	//AL UserState	
	IF e_US_AL > 0 THEN
		CASE e_US_AL OF
			1: cm_US1 := 1;
			2: cm_US2 := 1;
			3: cm_US3 := 1;
			4: cm_US4 := 1;
		END_CASE
	END_IF	
END_IF	

//IHT 
IF al_PCW_low OR al_IH_fail OR al_IH_overT OR al_SH_CW_overT OR al_IH_CW_overT THEN
	cm_IH := 0;
END_IF
					 
//H2 & SiH4 & NH3
IF is_AL THEN	
	cm_V01 := 0;// H2 Supply
	cm_V02 := 0;// H2 Supply
	cm_V03 := 0;//SiH4 Supply
	cm_V04 := 0;//NH3 Supply
END_IF

IF is_P01_overP_al THEN //둘다 닫아 자연스럽게 동자
	cm_V33_1 := 0;
	cm_V33_2 := 0;
END_IF

IF al_DOR OR wn_DOR THEN
	s_DOR_CNT := 0;
END_IF


//Buzzer Off Process
IF cm_BZ_UserStop OR P_di_RST.Q THEN
	IF n_BZ_Order[0] > 0 THEN
		n_BZ_Order[0] := 0; 
	ELSE
		n_BZ_Order[1] := 0;
	END_IF
	cm_BZ := 0;
	cm_BZ_UserStop := 0; 
END_IF

//Buzzer On Process
IF ing_Maint = 0 THEN	
	T1S_WN(PT:=T#1S);
	T1S_WN.IN :=  n_BZ_Order[0] + n_BZ_Order[1] = 1;
	IF T1S_WN.Q THEN //warning buzzer is 1sec cycle
		T1S_WN.IN := 0;
		cm_BZ := NOT cm_BZ;
	END_IF
	
	IF n_BZ_Order[0] + n_BZ_Order[1] >= 2 THEN
		cm_BZ := 1;
	END_IF
END_IF


//H2	
//IF al_N2_Low OR  al_H2_Low OR al_NH3_Low OR al_GC_H2_Leak OR al_RC_H2_Leak  THEN 
	//H2 Valve OFF - kjk??
	//cm_V27 := OFF;
//END_IF

//EMG_InductionPower
(*IF al_CW_IH_TempHi = ON THEN
	do_IH_Pow := OFF;
ELSE
	IF al_CHM_TempHi = ON THEN
		do_IH_Pow := OFF;
	ELSE
		IF al_GC_H2_Leak = ON THEN
			do_IH_Pow := OFF;
		ELSE
			IF al_RC_H2_Leak = ON THEN
				do_IH_Pow := OFF;
			ELSE
				do_IH_Pow := ON;	
			END_IF		
		END_IF		
	END_IF		
END_IF *)
END_ACTION

ACTION D_AL_Check:
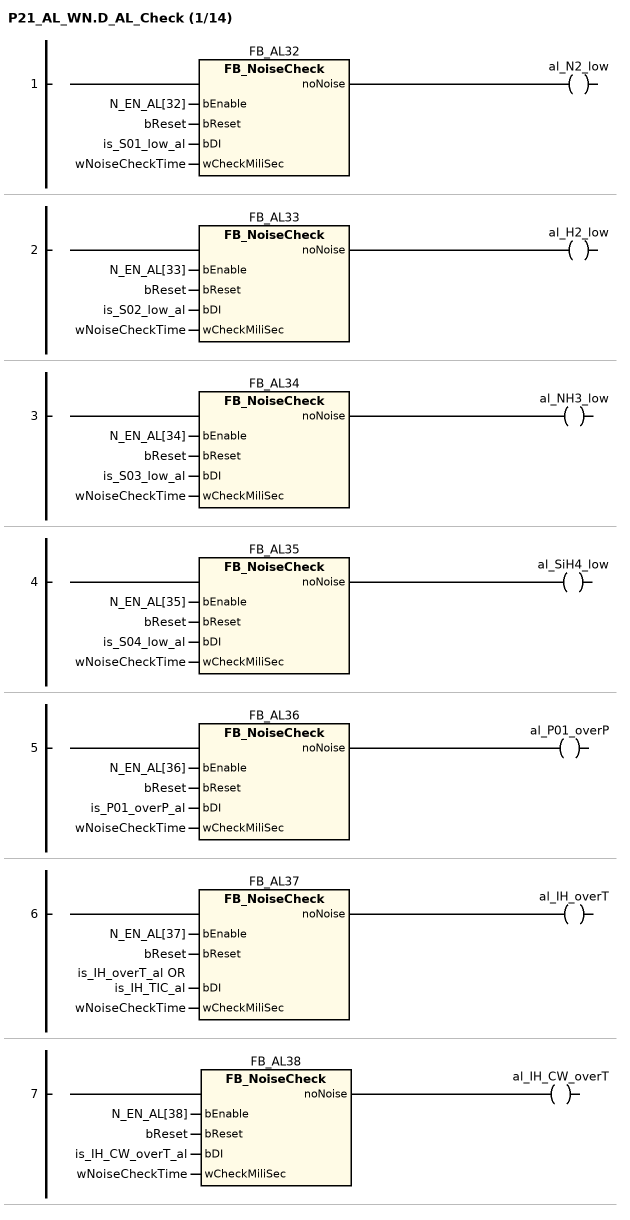
// NETWORK 1
FB_AL32(bEnable := N_EN_AL[32], bReset := bReset, bDI := is_S01_low_al, wCheckMiliSec := wNoiseCheckTime); // FB_NoiseCheck
al_N2_low := FB_AL32.noNoise;

// NETWORK 2
FB_AL33(bEnable := N_EN_AL[33], bReset := bReset, bDI := is_S02_low_al, wCheckMiliSec := wNoiseCheckTime); // FB_NoiseCheck
al_H2_low := FB_AL33.noNoise;

// NETWORK 3
FB_AL34(bEnable := N_EN_AL[34], bReset := bReset, bDI := is_S03_low_al, wCheckMiliSec := wNoiseCheckTime); // FB_NoiseCheck
al_NH3_low := FB_AL34.noNoise;

// NETWORK 4
FB_AL35(bEnable := N_EN_AL[35], bReset := bReset, bDI := is_S04_low_al, wCheckMiliSec := wNoiseCheckTime); // FB_NoiseCheck
al_SiH4_low := FB_AL35.noNoise;

// NETWORK 5
FB_AL36(bEnable := N_EN_AL[36], bReset := bReset, bDI := is_P01_overP_al, wCheckMiliSec := wNoiseCheckTime); // FB_NoiseCheck
al_P01_overP := FB_AL36.noNoise;

// NETWORK 6
FB_AL37(
    bEnable := N_EN_AL[37],
    bReset := bReset,
    bDI := is_IH_overT_al OR is_IH_TIC_al,
    wCheckMiliSec := wNoiseCheckTime); // FB_NoiseCheck
al_IH_overT := FB_AL37.noNoise;

// NETWORK 7
FB_AL38(bEnable := N_EN_AL[38], bReset := bReset, bDI := is_IH_CW_overT_al, wCheckMiliSec := wNoiseCheckTime); // FB_NoiseCheck
al_IH_CW_overT := FB_AL38.noNoise;

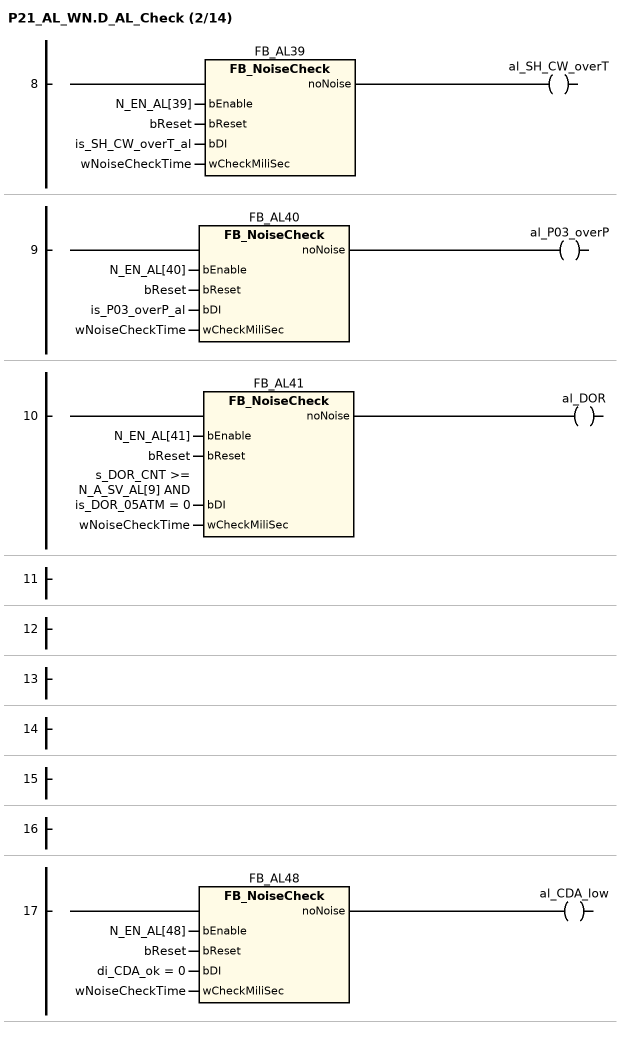
// NETWORK 8
FB_AL39(bEnable := N_EN_AL[39], bReset := bReset, bDI := is_SH_CW_overT_al, wCheckMiliSec := wNoiseCheckTime); // FB_NoiseCheck
al_SH_CW_overT := FB_AL39.noNoise;

// NETWORK 9
FB_AL40(bEnable := N_EN_AL[40], bReset := bReset, bDI := is_P03_overP_al, wCheckMiliSec := wNoiseCheckTime); // FB_NoiseCheck
al_P03_overP := FB_AL40.noNoise;

// NETWORK 10
FB_AL41(
    bEnable := N_EN_AL[41],
    bReset := bReset,
    bDI := s_DOR_CNT >= N_A_SV_AL[9] AND is_DOR_05ATM = 0,
    wCheckMiliSec := wNoiseCheckTime); // FB_NoiseCheck
al_DOR := FB_AL41.noNoise;

// NETWORK 11

// NETWORK 12

// NETWORK 13

// NETWORK 14

// NETWORK 15

// NETWORK 16

// NETWORK 17
FB_AL48(bEnable := N_EN_AL[48], bReset := bReset, bDI := di_CDA_ok = 0, wCheckMiliSec := wNoiseCheckTime); // FB_NoiseCheck
al_CDA_low := FB_AL48.noNoise;

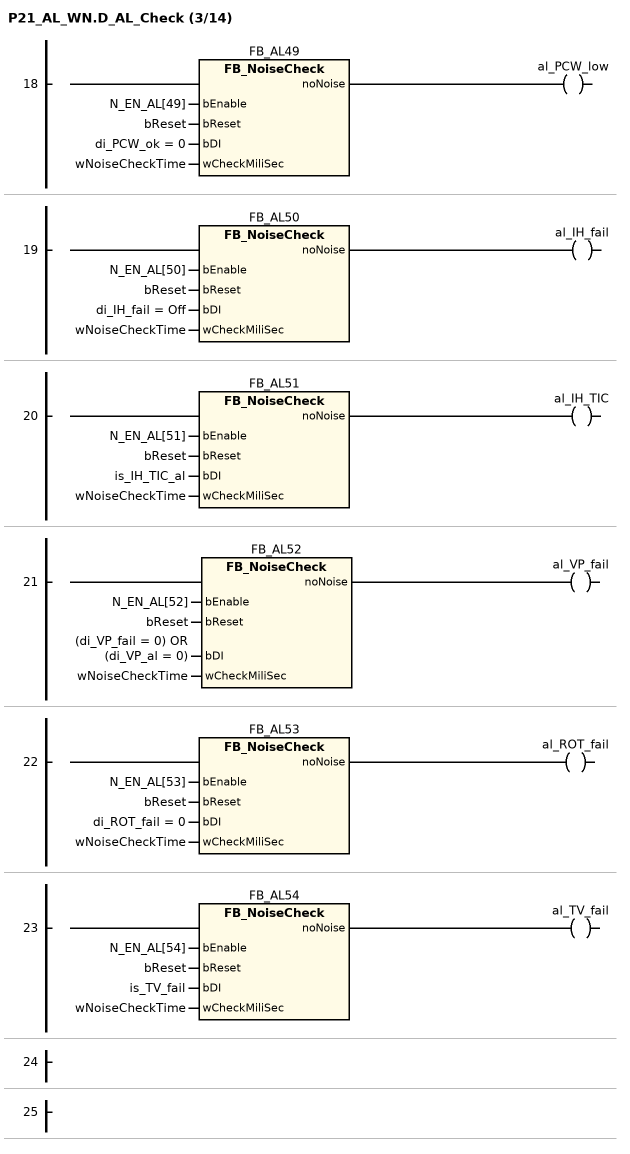
// NETWORK 18
FB_AL49(bEnable := N_EN_AL[49], bReset := bReset, bDI := di_PCW_ok = 0, wCheckMiliSec := wNoiseCheckTime); // FB_NoiseCheck
al_PCW_low := FB_AL49.noNoise;

// NETWORK 19
FB_AL50(bEnable := N_EN_AL[50], bReset := bReset, bDI := di_IH_fail = Off, wCheckMiliSec := wNoiseCheckTime); // FB_NoiseCheck
al_IH_fail := FB_AL50.noNoise;

// NETWORK 20
FB_AL51(bEnable := N_EN_AL[51], bReset := bReset, bDI := is_IH_TIC_al, wCheckMiliSec := wNoiseCheckTime); // FB_NoiseCheck
al_IH_TIC := FB_AL51.noNoise;

// NETWORK 21
FB_AL52(
    bEnable := N_EN_AL[52],
    bReset := bReset,
    bDI := (di_VP_fail = 0) OR (di_VP_al = 0),
    wCheckMiliSec := wNoiseCheckTime); // FB_NoiseCheck
al_VP_fail := FB_AL52.noNoise;

// NETWORK 22
FB_AL53(bEnable := N_EN_AL[53], bReset := bReset, bDI := di_ROT_fail = 0, wCheckMiliSec := wNoiseCheckTime); // FB_NoiseCheck
al_ROT_fail := FB_AL53.noNoise;

// NETWORK 23
FB_AL54(bEnable := N_EN_AL[54], bReset := bReset, bDI := is_TV_fail, wCheckMiliSec := wNoiseCheckTime); // FB_NoiseCheck
al_TV_fail := FB_AL54.noNoise;

// NETWORK 24

// NETWORK 25

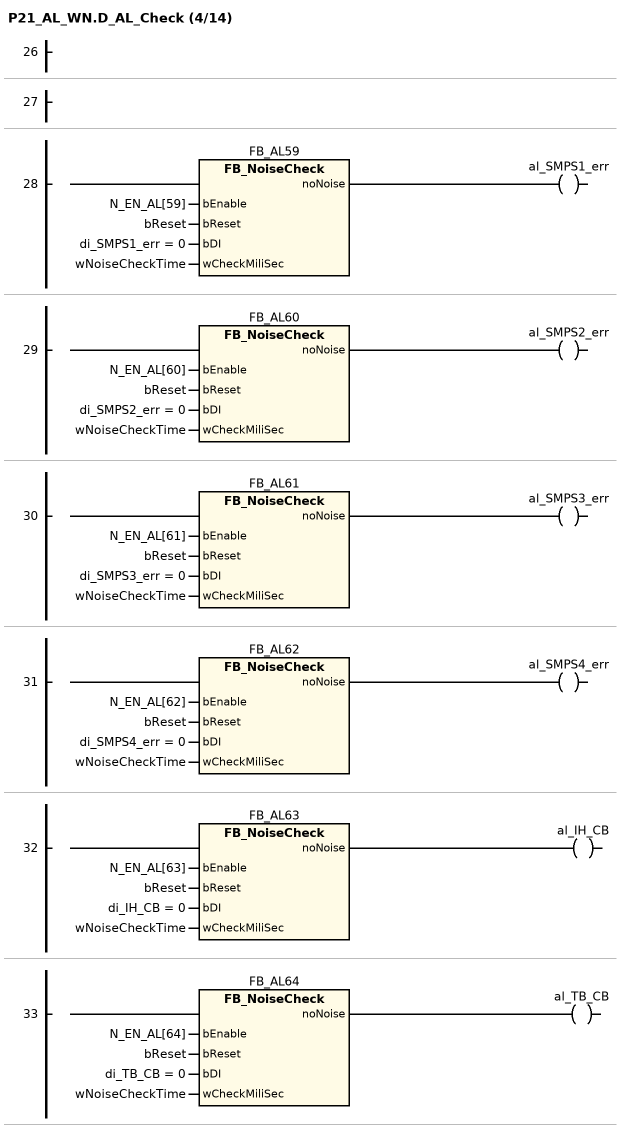
// NETWORK 26

// NETWORK 27

// NETWORK 28
FB_AL59(bEnable := N_EN_AL[59], bReset := bReset, bDI := di_SMPS1_err = 0, wCheckMiliSec := wNoiseCheckTime); // FB_NoiseCheck
al_SMPS1_err := FB_AL59.noNoise;

// NETWORK 29
FB_AL60(bEnable := N_EN_AL[60], bReset := bReset, bDI := di_SMPS2_err = 0, wCheckMiliSec := wNoiseCheckTime); // FB_NoiseCheck
al_SMPS2_err := FB_AL60.noNoise;

// NETWORK 30
FB_AL61(bEnable := N_EN_AL[61], bReset := bReset, bDI := di_SMPS3_err = 0, wCheckMiliSec := wNoiseCheckTime); // FB_NoiseCheck
al_SMPS3_err := FB_AL61.noNoise;

// NETWORK 31
FB_AL62(bEnable := N_EN_AL[62], bReset := bReset, bDI := di_SMPS4_err = 0, wCheckMiliSec := wNoiseCheckTime); // FB_NoiseCheck
al_SMPS4_err := FB_AL62.noNoise;

// NETWORK 32
FB_AL63(bEnable := N_EN_AL[63], bReset := bReset, bDI := di_IH_CB = 0, wCheckMiliSec := wNoiseCheckTime); // FB_NoiseCheck
al_IH_CB := FB_AL63.noNoise;

// NETWORK 33
FB_AL64(bEnable := N_EN_AL[64], bReset := bReset, bDI := di_TB_CB = 0, wCheckMiliSec := wNoiseCheckTime); // FB_NoiseCheck
al_TB_CB := FB_AL64.noNoise;

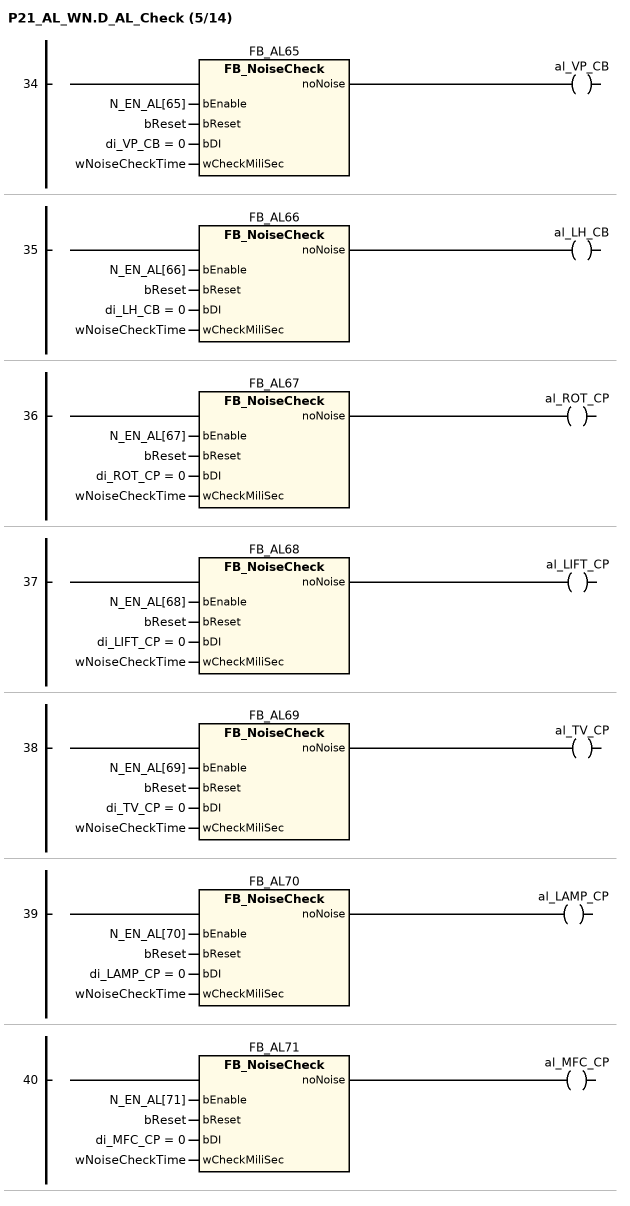
// NETWORK 34
FB_AL65(bEnable := N_EN_AL[65], bReset := bReset, bDI := di_VP_CB = 0, wCheckMiliSec := wNoiseCheckTime); // FB_NoiseCheck
al_VP_CB := FB_AL65.noNoise;

// NETWORK 35
FB_AL66(bEnable := N_EN_AL[66], bReset := bReset, bDI := di_LH_CB = 0, wCheckMiliSec := wNoiseCheckTime); // FB_NoiseCheck
al_LH_CB := FB_AL66.noNoise;

// NETWORK 36
FB_AL67(bEnable := N_EN_AL[67], bReset := bReset, bDI := di_ROT_CP = 0, wCheckMiliSec := wNoiseCheckTime); // FB_NoiseCheck
al_ROT_CP := FB_AL67.noNoise;

// NETWORK 37
FB_AL68(bEnable := N_EN_AL[68], bReset := bReset, bDI := di_LIFT_CP = 0, wCheckMiliSec := wNoiseCheckTime); // FB_NoiseCheck
al_LIFT_CP := FB_AL68.noNoise;

// NETWORK 38
FB_AL69(bEnable := N_EN_AL[69], bReset := bReset, bDI := di_TV_CP = 0, wCheckMiliSec := wNoiseCheckTime); // FB_NoiseCheck
al_TV_CP := FB_AL69.noNoise;

// NETWORK 39
FB_AL70(bEnable := N_EN_AL[70], bReset := bReset, bDI := di_LAMP_CP = 0, wCheckMiliSec := wNoiseCheckTime); // FB_NoiseCheck
al_LAMP_CP := FB_AL70.noNoise;

// NETWORK 40
FB_AL71(bEnable := N_EN_AL[71], bReset := bReset, bDI := di_MFC_CP = 0, wCheckMiliSec := wNoiseCheckTime); // FB_NoiseCheck
al_MFC_CP := FB_AL71.noNoise;

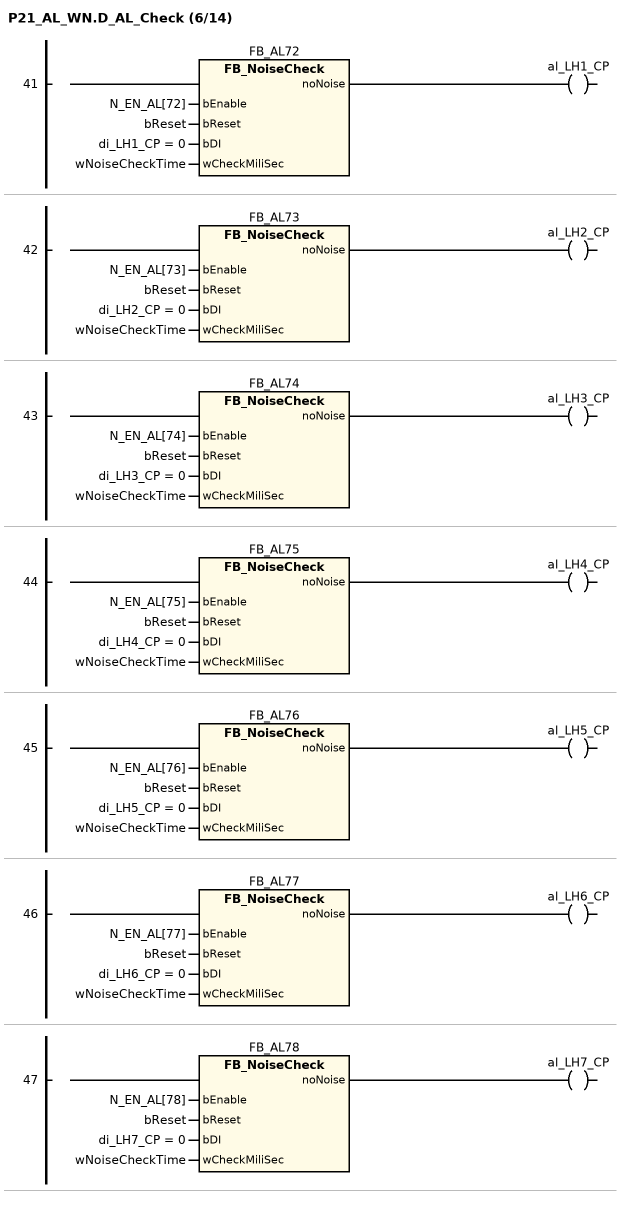
// NETWORK 41
FB_AL72(bEnable := N_EN_AL[72], bReset := bReset, bDI := di_LH1_CP = 0, wCheckMiliSec := wNoiseCheckTime); // FB_NoiseCheck
al_LH1_CP := FB_AL72.noNoise;

// NETWORK 42
FB_AL73(bEnable := N_EN_AL[73], bReset := bReset, bDI := di_LH2_CP = 0, wCheckMiliSec := wNoiseCheckTime); // FB_NoiseCheck
al_LH2_CP := FB_AL73.noNoise;

// NETWORK 43
FB_AL74(bEnable := N_EN_AL[74], bReset := bReset, bDI := di_LH3_CP = 0, wCheckMiliSec := wNoiseCheckTime); // FB_NoiseCheck
al_LH3_CP := FB_AL74.noNoise;

// NETWORK 44
FB_AL75(bEnable := N_EN_AL[75], bReset := bReset, bDI := di_LH4_CP = 0, wCheckMiliSec := wNoiseCheckTime); // FB_NoiseCheck
al_LH4_CP := FB_AL75.noNoise;

// NETWORK 45
FB_AL76(bEnable := N_EN_AL[76], bReset := bReset, bDI := di_LH5_CP = 0, wCheckMiliSec := wNoiseCheckTime); // FB_NoiseCheck
al_LH5_CP := FB_AL76.noNoise;

// NETWORK 46
FB_AL77(bEnable := N_EN_AL[77], bReset := bReset, bDI := di_LH6_CP = 0, wCheckMiliSec := wNoiseCheckTime); // FB_NoiseCheck
al_LH6_CP := FB_AL77.noNoise;

// NETWORK 47
FB_AL78(bEnable := N_EN_AL[78], bReset := bReset, bDI := di_LH7_CP = 0, wCheckMiliSec := wNoiseCheckTime); // FB_NoiseCheck
al_LH7_CP := FB_AL78.noNoise;

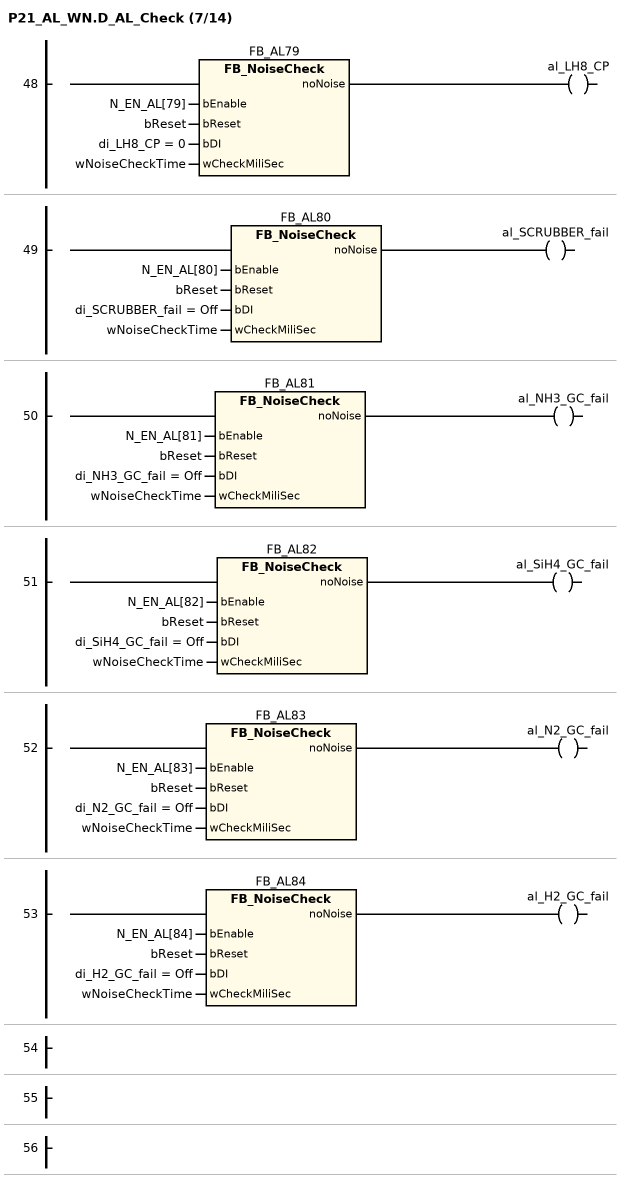
// NETWORK 48
FB_AL79(bEnable := N_EN_AL[79], bReset := bReset, bDI := di_LH8_CP = 0, wCheckMiliSec := wNoiseCheckTime); // FB_NoiseCheck
al_LH8_CP := FB_AL79.noNoise;

// NETWORK 49
FB_AL80(
    bEnable := N_EN_AL[80],
    bReset := bReset,
    bDI := di_SCRUBBER_fail = Off,
    wCheckMiliSec := wNoiseCheckTime); // FB_NoiseCheck
al_SCRUBBER_fail := FB_AL80.noNoise;

// NETWORK 50
FB_AL81(
    bEnable := N_EN_AL[81],
    bReset := bReset,
    bDI := di_NH3_GC_fail = Off,
    wCheckMiliSec := wNoiseCheckTime); // FB_NoiseCheck
al_NH3_GC_fail := FB_AL81.noNoise;

// NETWORK 51
FB_AL82(
    bEnable := N_EN_AL[82],
    bReset := bReset,
    bDI := di_SiH4_GC_fail = Off,
    wCheckMiliSec := wNoiseCheckTime); // FB_NoiseCheck
al_SiH4_GC_fail := FB_AL82.noNoise;

// NETWORK 52
FB_AL83(
    bEnable := N_EN_AL[83],
    bReset := bReset,
    bDI := di_N2_GC_fail = Off,
    wCheckMiliSec := wNoiseCheckTime); // FB_NoiseCheck
al_N2_GC_fail := FB_AL83.noNoise;

// NETWORK 53
FB_AL84(
    bEnable := N_EN_AL[84],
    bReset := bReset,
    bDI := di_H2_GC_fail = Off,
    wCheckMiliSec := wNoiseCheckTime); // FB_NoiseCheck
al_H2_GC_fail := FB_AL84.noNoise;

// NETWORK 54

// NETWORK 55

// NETWORK 56

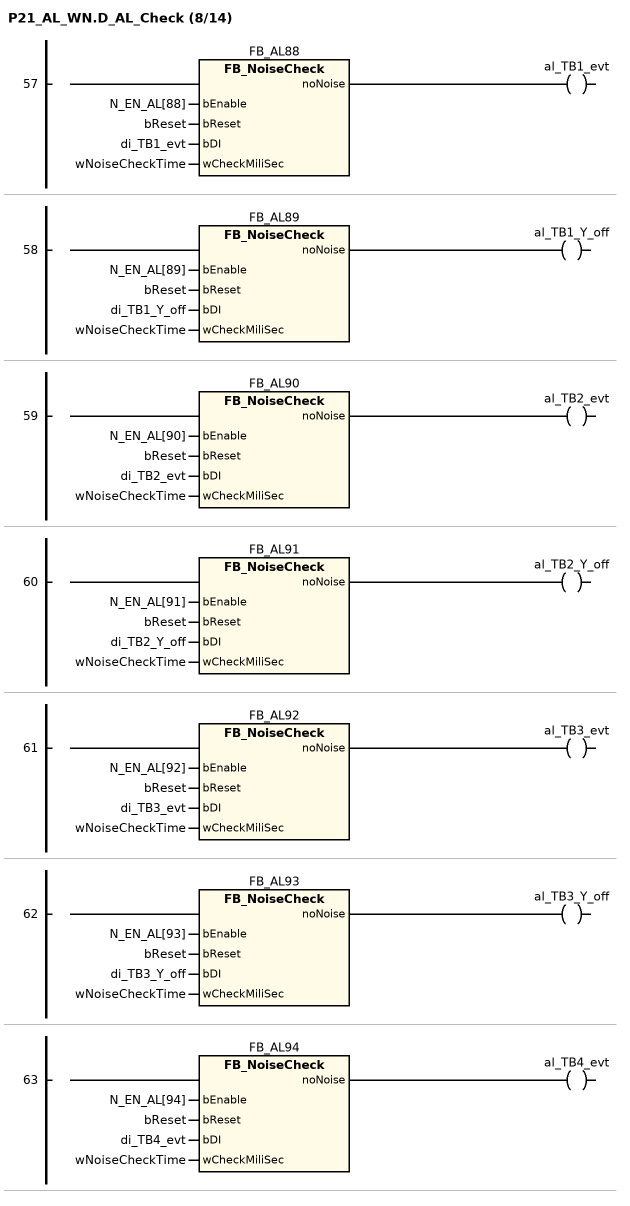
// NETWORK 57
FB_AL88(bEnable := N_EN_AL[88], bReset := bReset, bDI := di_TB1_evt, wCheckMiliSec := wNoiseCheckTime); // FB_NoiseCheck
al_TB1_evt := FB_AL88.noNoise;

// NETWORK 58
FB_AL89(bEnable := N_EN_AL[89], bReset := bReset, bDI := di_TB1_Y_off, wCheckMiliSec := wNoiseCheckTime); // FB_NoiseCheck
al_TB1_Y_off := FB_AL89.noNoise;

// NETWORK 59
FB_AL90(bEnable := N_EN_AL[90], bReset := bReset, bDI := di_TB2_evt, wCheckMiliSec := wNoiseCheckTime); // FB_NoiseCheck
al_TB2_evt := FB_AL90.noNoise;

// NETWORK 60
FB_AL91(bEnable := N_EN_AL[91], bReset := bReset, bDI := di_TB2_Y_off, wCheckMiliSec := wNoiseCheckTime); // FB_NoiseCheck
al_TB2_Y_off := FB_AL91.noNoise;

// NETWORK 61
FB_AL92(bEnable := N_EN_AL[92], bReset := bReset, bDI := di_TB3_evt, wCheckMiliSec := wNoiseCheckTime); // FB_NoiseCheck
al_TB3_evt := FB_AL92.noNoise;

// NETWORK 62
FB_AL93(bEnable := N_EN_AL[93], bReset := bReset, bDI := di_TB3_Y_off, wCheckMiliSec := wNoiseCheckTime); // FB_NoiseCheck
al_TB3_Y_off := FB_AL93.noNoise;

// NETWORK 63
FB_AL94(bEnable := N_EN_AL[94], bReset := bReset, bDI := di_TB4_evt, wCheckMiliSec := wNoiseCheckTime); // FB_NoiseCheck
al_TB4_evt := FB_AL94.noNoise;

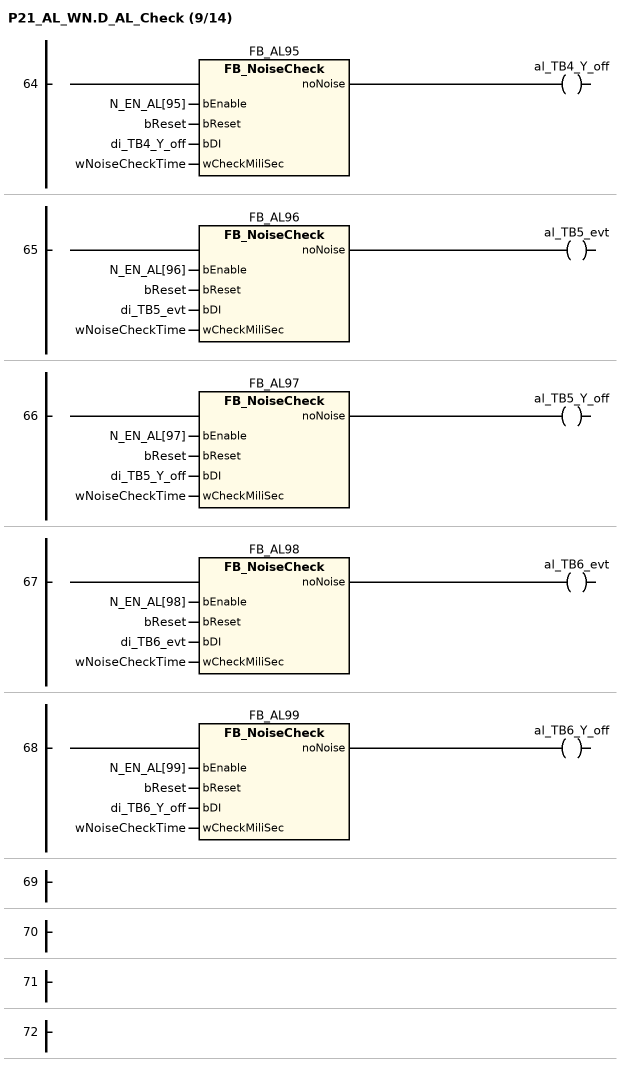
// NETWORK 64
FB_AL95(bEnable := N_EN_AL[95], bReset := bReset, bDI := di_TB4_Y_off, wCheckMiliSec := wNoiseCheckTime); // FB_NoiseCheck
al_TB4_Y_off := FB_AL95.noNoise;

// NETWORK 65
FB_AL96(bEnable := N_EN_AL[96], bReset := bReset, bDI := di_TB5_evt, wCheckMiliSec := wNoiseCheckTime); // FB_NoiseCheck
al_TB5_evt := FB_AL96.noNoise;

// NETWORK 66
FB_AL97(bEnable := N_EN_AL[97], bReset := bReset, bDI := di_TB5_Y_off, wCheckMiliSec := wNoiseCheckTime); // FB_NoiseCheck
al_TB5_Y_off := FB_AL97.noNoise;

// NETWORK 67
FB_AL98(bEnable := N_EN_AL[98], bReset := bReset, bDI := di_TB6_evt, wCheckMiliSec := wNoiseCheckTime); // FB_NoiseCheck
al_TB6_evt := FB_AL98.noNoise;

// NETWORK 68
FB_AL99(bEnable := N_EN_AL[99], bReset := bReset, bDI := di_TB6_Y_off, wCheckMiliSec := wNoiseCheckTime); // FB_NoiseCheck
al_TB6_Y_off := FB_AL99.noNoise;

// NETWORK 69

// NETWORK 70

// NETWORK 71

// NETWORK 72

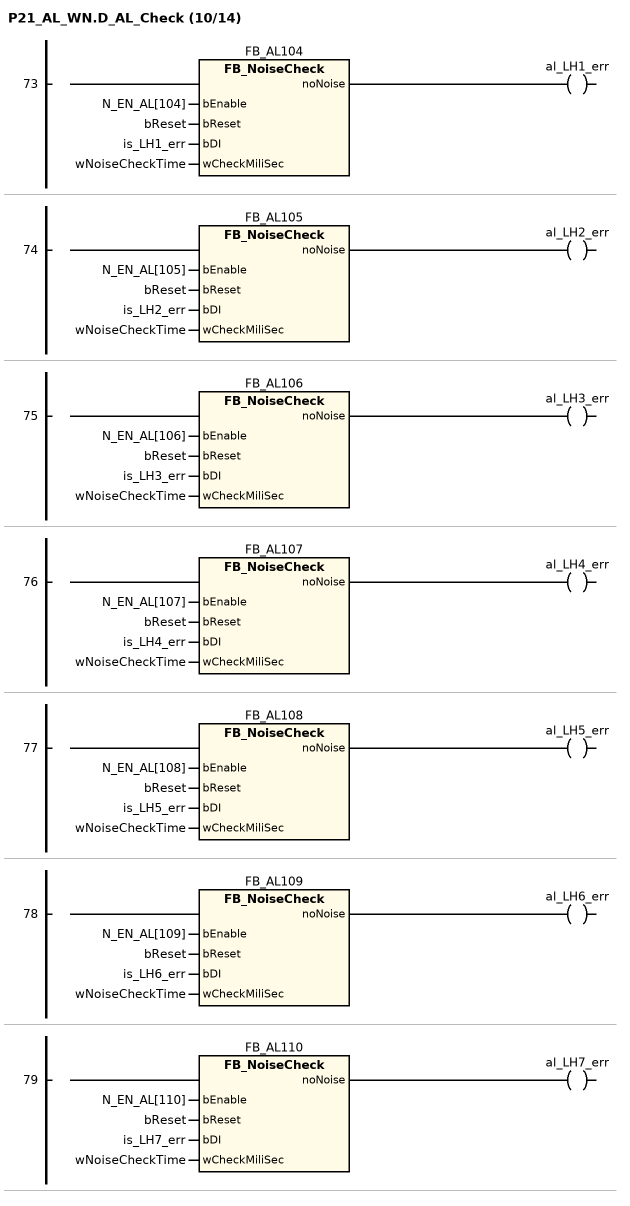
// NETWORK 73
FB_AL104(bEnable := N_EN_AL[104], bReset := bReset, bDI := is_LH1_err, wCheckMiliSec := wNoiseCheckTime); // FB_NoiseCheck
al_LH1_err := FB_AL104.noNoise;

// NETWORK 74
FB_AL105(bEnable := N_EN_AL[105], bReset := bReset, bDI := is_LH2_err, wCheckMiliSec := wNoiseCheckTime); // FB_NoiseCheck
al_LH2_err := FB_AL105.noNoise;

// NETWORK 75
FB_AL106(bEnable := N_EN_AL[106], bReset := bReset, bDI := is_LH3_err, wCheckMiliSec := wNoiseCheckTime); // FB_NoiseCheck
al_LH3_err := FB_AL106.noNoise;

// NETWORK 76
FB_AL107(bEnable := N_EN_AL[107], bReset := bReset, bDI := is_LH4_err, wCheckMiliSec := wNoiseCheckTime); // FB_NoiseCheck
al_LH4_err := FB_AL107.noNoise;

// NETWORK 77
FB_AL108(bEnable := N_EN_AL[108], bReset := bReset, bDI := is_LH5_err, wCheckMiliSec := wNoiseCheckTime); // FB_NoiseCheck
al_LH5_err := FB_AL108.noNoise;

// NETWORK 78
FB_AL109(bEnable := N_EN_AL[109], bReset := bReset, bDI := is_LH6_err, wCheckMiliSec := wNoiseCheckTime); // FB_NoiseCheck
al_LH6_err := FB_AL109.noNoise;

// NETWORK 79
FB_AL110(bEnable := N_EN_AL[110], bReset := bReset, bDI := is_LH7_err, wCheckMiliSec := wNoiseCheckTime); // FB_NoiseCheck
al_LH7_err := FB_AL110.noNoise;

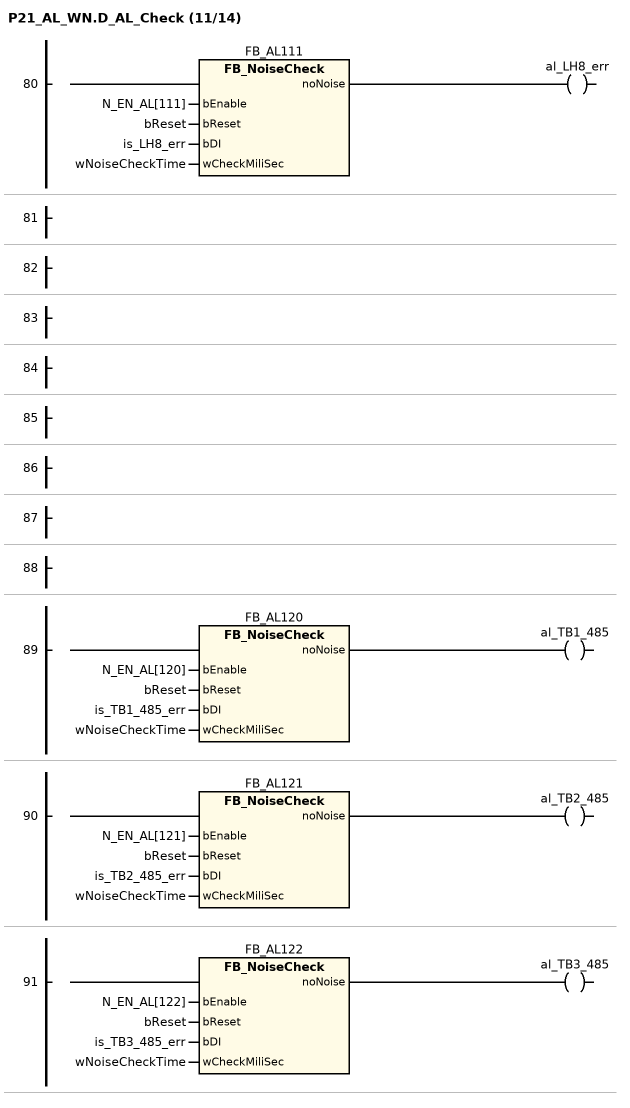
// NETWORK 80
FB_AL111(bEnable := N_EN_AL[111], bReset := bReset, bDI := is_LH8_err, wCheckMiliSec := wNoiseCheckTime); // FB_NoiseCheck
al_LH8_err := FB_AL111.noNoise;

// NETWORK 81

// NETWORK 82

// NETWORK 83

// NETWORK 84

// NETWORK 85

// NETWORK 86

// NETWORK 87

// NETWORK 88

// NETWORK 89
FB_AL120(bEnable := N_EN_AL[120], bReset := bReset, bDI := is_TB1_485_err, wCheckMiliSec := wNoiseCheckTime); // FB_NoiseCheck
al_TB1_485 := FB_AL120.noNoise;

// NETWORK 90
FB_AL121(bEnable := N_EN_AL[121], bReset := bReset, bDI := is_TB2_485_err, wCheckMiliSec := wNoiseCheckTime); // FB_NoiseCheck
al_TB2_485 := FB_AL121.noNoise;

// NETWORK 91
FB_AL122(bEnable := N_EN_AL[122], bReset := bReset, bDI := is_TB3_485_err, wCheckMiliSec := wNoiseCheckTime); // FB_NoiseCheck
al_TB3_485 := FB_AL122.noNoise;

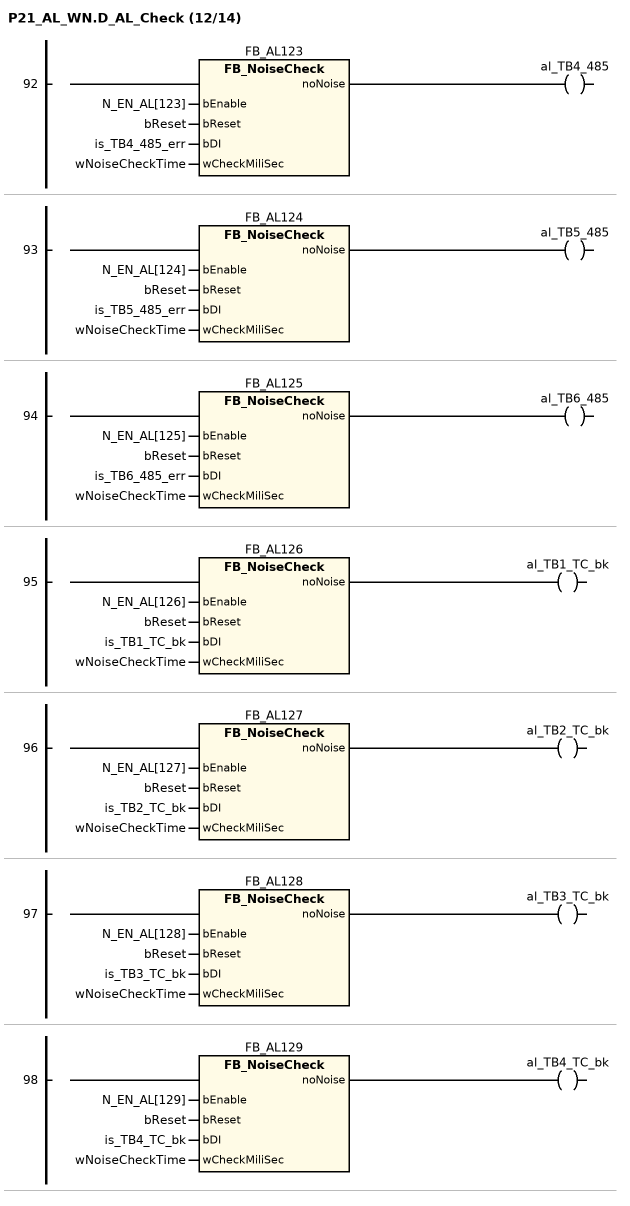
// NETWORK 92
FB_AL123(bEnable := N_EN_AL[123], bReset := bReset, bDI := is_TB4_485_err, wCheckMiliSec := wNoiseCheckTime); // FB_NoiseCheck
al_TB4_485 := FB_AL123.noNoise;

// NETWORK 93
FB_AL124(bEnable := N_EN_AL[124], bReset := bReset, bDI := is_TB5_485_err, wCheckMiliSec := wNoiseCheckTime); // FB_NoiseCheck
al_TB5_485 := FB_AL124.noNoise;

// NETWORK 94
FB_AL125(bEnable := N_EN_AL[125], bReset := bReset, bDI := is_TB6_485_err, wCheckMiliSec := wNoiseCheckTime); // FB_NoiseCheck
al_TB6_485 := FB_AL125.noNoise;

// NETWORK 95
FB_AL126(bEnable := N_EN_AL[126], bReset := bReset, bDI := is_TB1_TC_bk, wCheckMiliSec := wNoiseCheckTime); // FB_NoiseCheck
al_TB1_TC_bk := FB_AL126.noNoise;

// NETWORK 96
FB_AL127(bEnable := N_EN_AL[127], bReset := bReset, bDI := is_TB2_TC_bk, wCheckMiliSec := wNoiseCheckTime); // FB_NoiseCheck
al_TB2_TC_bk := FB_AL127.noNoise;

// NETWORK 97
FB_AL128(bEnable := N_EN_AL[128], bReset := bReset, bDI := is_TB3_TC_bk, wCheckMiliSec := wNoiseCheckTime); // FB_NoiseCheck
al_TB3_TC_bk := FB_AL128.noNoise;

// NETWORK 98
FB_AL129(bEnable := N_EN_AL[129], bReset := bReset, bDI := is_TB4_TC_bk, wCheckMiliSec := wNoiseCheckTime); // FB_NoiseCheck
al_TB4_TC_bk := FB_AL129.noNoise;

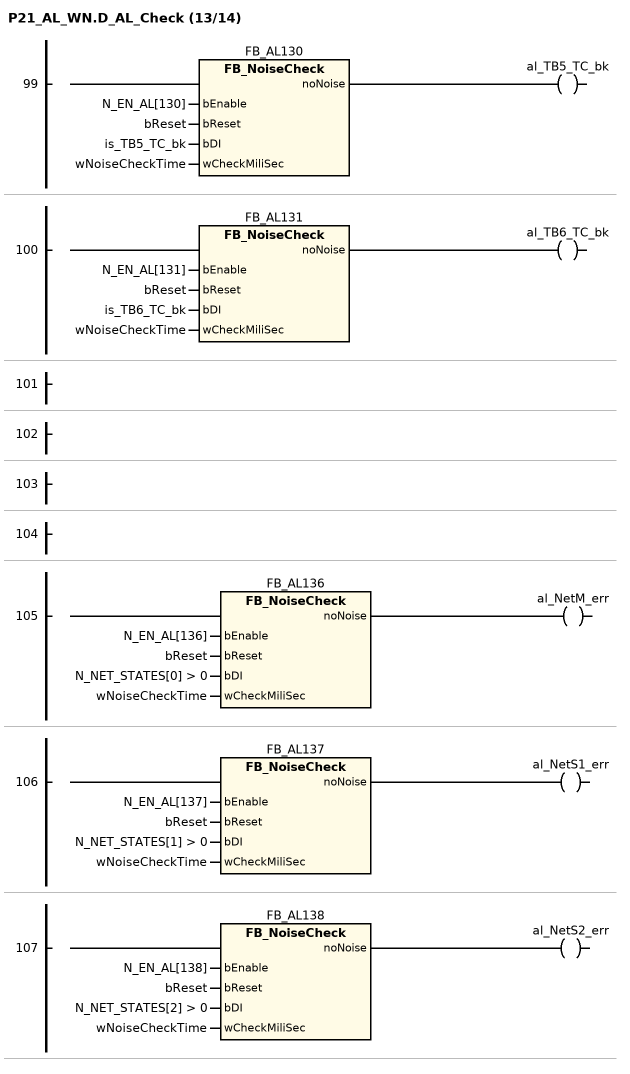
// NETWORK 99
FB_AL130(bEnable := N_EN_AL[130], bReset := bReset, bDI := is_TB5_TC_bk, wCheckMiliSec := wNoiseCheckTime); // FB_NoiseCheck
al_TB5_TC_bk := FB_AL130.noNoise;

// NETWORK 100
FB_AL131(bEnable := N_EN_AL[131], bReset := bReset, bDI := is_TB6_TC_bk, wCheckMiliSec := wNoiseCheckTime); // FB_NoiseCheck
al_TB6_TC_bk := FB_AL131.noNoise;

// NETWORK 101

// NETWORK 102

// NETWORK 103

// NETWORK 104

// NETWORK 105
FB_AL136(
    bEnable := N_EN_AL[136],
    bReset := bReset,
    bDI := N_NET_STATES[0] > 0,
    wCheckMiliSec := wNoiseCheckTime); // FB_NoiseCheck
al_NetM_err := FB_AL136.noNoise;

// NETWORK 106
FB_AL137(
    bEnable := N_EN_AL[137],
    bReset := bReset,
    bDI := N_NET_STATES[1] > 0,
    wCheckMiliSec := wNoiseCheckTime); // FB_NoiseCheck
al_NetS1_err := FB_AL137.noNoise;

// NETWORK 107
FB_AL138(
    bEnable := N_EN_AL[138],
    bReset := bReset,
    bDI := N_NET_STATES[2] > 0,
    wCheckMiliSec := wNoiseCheckTime); // FB_NoiseCheck
al_NetS2_err := FB_AL138.noNoise;

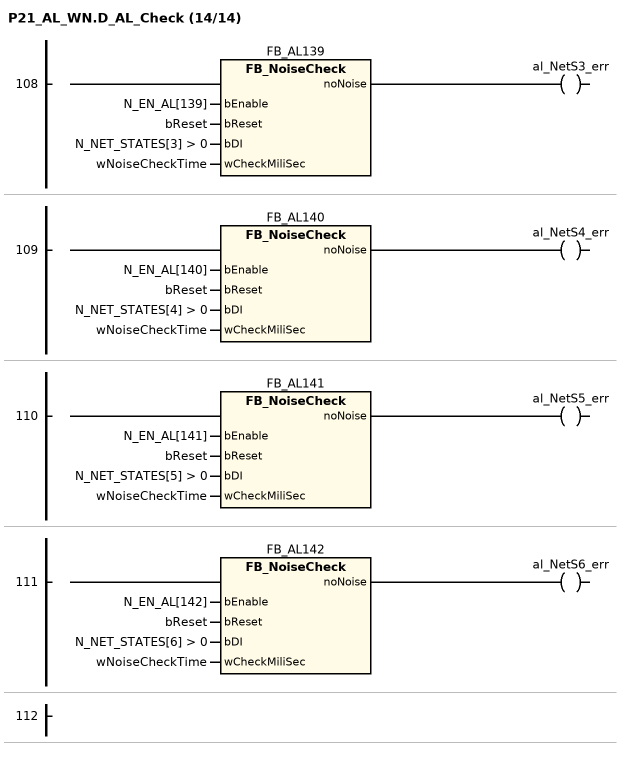
// NETWORK 108
FB_AL139(
    bEnable := N_EN_AL[139],
    bReset := bReset,
    bDI := N_NET_STATES[3] > 0,
    wCheckMiliSec := wNoiseCheckTime); // FB_NoiseCheck
al_NetS3_err := FB_AL139.noNoise;

// NETWORK 109
FB_AL140(
    bEnable := N_EN_AL[140],
    bReset := bReset,
    bDI := N_NET_STATES[4] > 0,
    wCheckMiliSec := wNoiseCheckTime); // FB_NoiseCheck
al_NetS4_err := FB_AL140.noNoise;

// NETWORK 110
FB_AL141(
    bEnable := N_EN_AL[141],
    bReset := bReset,
    bDI := N_NET_STATES[5] > 0,
    wCheckMiliSec := wNoiseCheckTime); // FB_NoiseCheck
al_NetS5_err := FB_AL141.noNoise;

// NETWORK 111
FB_AL142(
    bEnable := N_EN_AL[142],
    bReset := bReset,
    bDI := N_NET_STATES[6] > 0,
    wCheckMiliSec := wNoiseCheckTime); // FB_NoiseCheck
al_NetS6_err := FB_AL142.noNoise;

// NETWORK 112
END_ACTION

ACTION D_WN_Check:
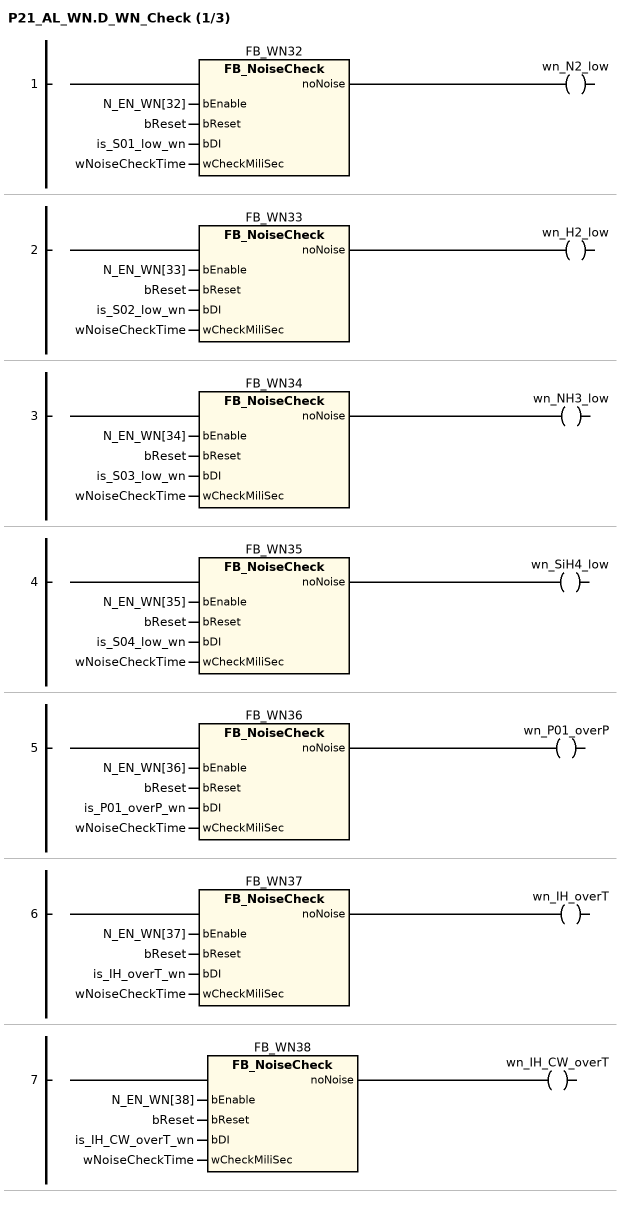
// NETWORK 1
FB_WN32(bEnable := N_EN_WN[32], bReset := bReset, bDI := is_S01_low_wn, wCheckMiliSec := wNoiseCheckTime); // FB_NoiseCheck
wn_N2_low := FB_WN32.noNoise;

// NETWORK 2
FB_WN33(bEnable := N_EN_WN[33], bReset := bReset, bDI := is_S02_low_wn, wCheckMiliSec := wNoiseCheckTime); // FB_NoiseCheck
wn_H2_low := FB_WN33.noNoise;

// NETWORK 3
FB_WN34(bEnable := N_EN_WN[34], bReset := bReset, bDI := is_S03_low_wn, wCheckMiliSec := wNoiseCheckTime); // FB_NoiseCheck
wn_NH3_low := FB_WN34.noNoise;

// NETWORK 4
FB_WN35(bEnable := N_EN_WN[35], bReset := bReset, bDI := is_S04_low_wn, wCheckMiliSec := wNoiseCheckTime); // FB_NoiseCheck
wn_SiH4_low := FB_WN35.noNoise;

// NETWORK 5
FB_WN36(bEnable := N_EN_WN[36], bReset := bReset, bDI := is_P01_overP_wn, wCheckMiliSec := wNoiseCheckTime); // FB_NoiseCheck
wn_P01_overP := FB_WN36.noNoise;

// NETWORK 6
FB_WN37(bEnable := N_EN_WN[37], bReset := bReset, bDI := is_IH_overT_wn, wCheckMiliSec := wNoiseCheckTime); // FB_NoiseCheck
wn_IH_overT := FB_WN37.noNoise;

// NETWORK 7
FB_WN38(bEnable := N_EN_WN[38], bReset := bReset, bDI := is_IH_CW_overT_wn, wCheckMiliSec := wNoiseCheckTime); // FB_NoiseCheck
wn_IH_CW_overT := FB_WN38.noNoise;

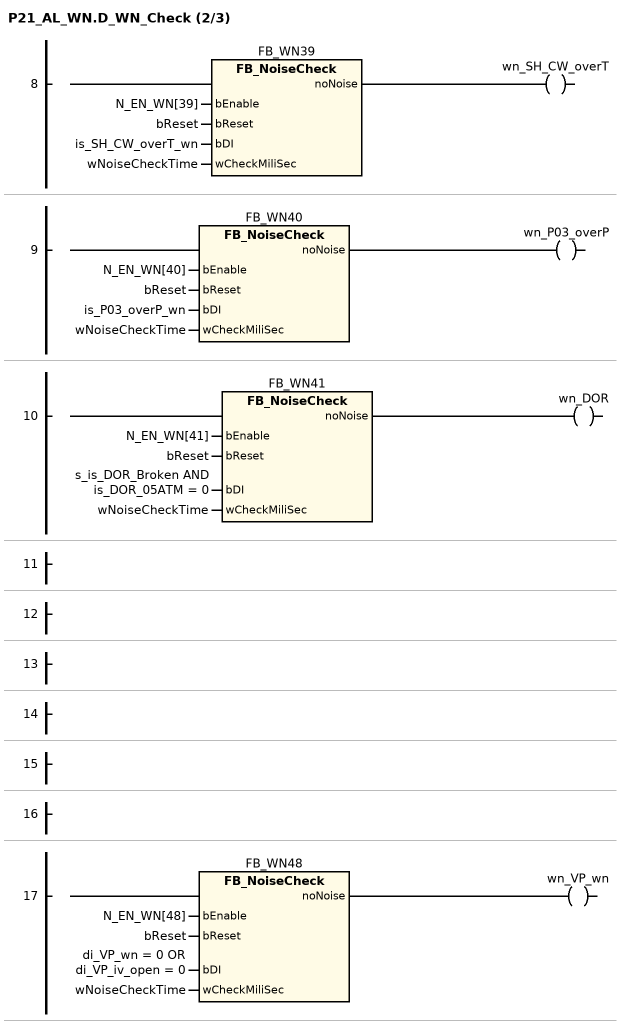
// NETWORK 8
FB_WN39(bEnable := N_EN_WN[39], bReset := bReset, bDI := is_SH_CW_overT_wn, wCheckMiliSec := wNoiseCheckTime); // FB_NoiseCheck
wn_SH_CW_overT := FB_WN39.noNoise;

// NETWORK 9
FB_WN40(bEnable := N_EN_WN[40], bReset := bReset, bDI := is_P03_overP_wn, wCheckMiliSec := wNoiseCheckTime); // FB_NoiseCheck
wn_P03_overP := FB_WN40.noNoise;

// NETWORK 10
FB_WN41(
    bEnable := N_EN_WN[41],
    bReset := bReset,
    bDI := s_is_DOR_Broken AND is_DOR_05ATM = 0,
    wCheckMiliSec := wNoiseCheckTime); // FB_NoiseCheck
wn_DOR := FB_WN41.noNoise;

// NETWORK 11

// NETWORK 12

// NETWORK 13

// NETWORK 14

// NETWORK 15

// NETWORK 16

// NETWORK 17
FB_WN48(
    bEnable := N_EN_WN[48],
    bReset := bReset,
    bDI := di_VP_wn = 0 OR di_VP_iv_open = 0,
    wCheckMiliSec := wNoiseCheckTime); // FB_NoiseCheck
wn_VP_wn := FB_WN48.noNoise;

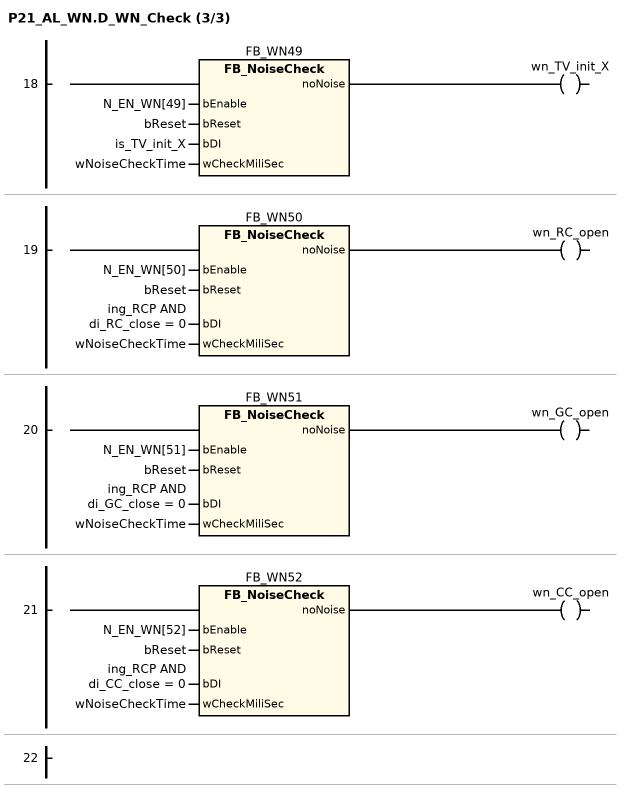
// NETWORK 18
FB_WN49(bEnable := N_EN_WN[49], bReset := bReset, bDI := is_TV_init_X, wCheckMiliSec := wNoiseCheckTime); // FB_NoiseCheck
wn_TV_init_X := FB_WN49.noNoise;

// NETWORK 19
FB_WN50(
    bEnable := N_EN_WN[50],
    bReset := bReset,
    bDI := ing_RCP AND di_RC_close = 0,
    wCheckMiliSec := wNoiseCheckTime); // FB_NoiseCheck
wn_RC_open := FB_WN50.noNoise;

// NETWORK 20
FB_WN51(
    bEnable := N_EN_WN[51],
    bReset := bReset,
    bDI := ing_RCP AND di_GC_close = 0,
    wCheckMiliSec := wNoiseCheckTime); // FB_NoiseCheck
wn_GC_open := FB_WN51.noNoise;

// NETWORK 21
FB_WN52(
    bEnable := N_EN_WN[52],
    bReset := bReset,
    bDI := ing_RCP AND di_CC_close = 0,
    wCheckMiliSec := wNoiseCheckTime); // FB_NoiseCheck
wn_CC_open := FB_WN52.noNoise;

// NETWORK 22
END_ACTION

END_PROGRAM

// ---- POUs/MR_PRG/P22_RCP_Ctrl.TcPOU
PROGRAM P22_RCP_Ctrl
VAR	
	p_Start, p_EMS: R_TRIG;
	nCase: INT;
	T_Ramp, T_Hold, T_Pause, T_Run: TON;	
	PT_MAX: TIME := T#4294967295MS;
	PT_RAMP, PT_HOLD: TIME;
	ET_RAMP, ET_HOLD, ET_RUN, ET_Pause: TIME;
	PT_RAMP_REMAIN, PT_HOLD_REMAIN: TIME;
	ET_RAMP_RUN, ET_HOLD_RUN: TIME;
		
	nLoop, nJump: INT;
    stepIdx: INT;
	nPauseStep: INT;	
	idx: INT;	
	
	nLoop_Cnt: INT;	
	jumpStart: INT;
	jumpEnd: INT;	
	
	SecScale: REAL;
	i_RUN_TM: DINT;
	i_RUN_TM_OLD: DINT;
END_VAR

//Timer
T_Ramp(PT:= PT_RAMP, ET=> ET_RAMP);  (*램핑 타이머 *)
T_Hold(PT:= PT_HOLD, ET=> ET_HOLD);  (*홀딩 타이머 *)
T_RUN(IN:= s_EN_EXE_RCP, PT:= PT_MAX , ET=> ET_RUN);  (*홀딩 타이머 *)
T_Pause(IN:= s_is_RCP_pause, PT:= PT_MAX, ET=> ET_Pause);

p_Start(CLK:= s_EN_EXE_RCP);
p_EMS(CLK:= (nCase > 0 AND s_EN_EXE_RCP = 0) OR is_AL);

IF p_Start.Q THEN
	nCase := 1;
END_IF

IF p_EMS.Q THEN
	s_EN_EXE_RCP := 0;
	nCase := 0;
END_IF

//IF EN_RUN_RCP THEN
IF nCase = 1 THEN (*Initial Setting*)
	cm_TV_run := 1;
	cm_ROT := 1;
	pv_RCP_RUN_ET := 0;
	pv_STEP_RTM := 0;
	pv_STEP_HTM := 0;
	pv_RCP_PAUSE_ET := 0;
	pv_STEP_LOOP := 0;
	sv_STEP_JUMP := 0;
	cm_RCP_pause := 0;
	cm_RCP_restart := 0;
	cm_RCP_skip := 0;
	is_RCP_ended := 0;
	s_is_RCP_pause := 0;
	nLoop := 0;
	stepIdx	:= 0;
	SecScale := UINT_TO_REAL(e_RTM_UNIT);						
	nCase := 10;		
END_IF

//Data Exchange
IF nCase = 10 THEN	
	//Ramp & Hold Time Init
	sv_STEP_RTM := UINT_TO_REAL(N_RCP_RTM[stepIdx]);
	sv_STEP_HTM := UINT_TO_REAL(N_RCP_HTM[stepIdx]); 
	PT_RAMP := REAL_TO_TIME(sv_STEP_RTM * SecScale);//1000;
	PT_HOLD := REAL_TO_TIME(sv_STEP_HTM * SecScale);//1000;    
    PT_RAMP_REMAIN := T#0MS;
	PT_HOLD_REMAIN := T#0MS;
	ET_RAMP_RUN := T#0MS;
	ET_HOLD_RUN := T#0MS;
		
	FOR idx := 0 TO 29 DO		
		IF N_EN_RCP_RAMP[idx] THEN	
			N_TSV_RTM[idx * 2 + 1] := sv_STEP_RTM;
		ELSE
			N_TSV_RTM[idx * 2 + 1] := 0;	
		END_IF				   			
	END_FOR  

	(*Analog value input *)
	tsv_M01	:= N_RCP_M01[stepIdx];	tsv_M02	:= N_RCP_M02[stepIdx];							
	tsv_M03	:= N_RCP_M03[stepIdx];	tsv_M04	:= N_RCP_M04[stepIdx];
	tsv_M05	:= N_RCP_M05[stepIdx];	tsv_M06	:= N_RCP_M06[stepIdx];
	tsv_M07	:= N_RCP_M07[stepIdx];	tsv_M08	:= N_RCP_M08[stepIdx];
	tsv_M09	:= N_RCP_M09[stepIdx];	tsv_M10	:= N_RCP_M10[stepIdx];
	tsv_M11	:= N_RCP_M11[stepIdx];	tsv_M12	:= N_RCP_M12[stepIdx];
	tsv_M13	:= N_RCP_M13[stepIdx];	tsv_M14	:= N_RCP_M14[stepIdx];
	tsv_M15	:= N_RCP_M15[stepIdx];	tsv_M16	:= N_RCP_M16[stepIdx];
	tsv_M17	:= N_RCP_M17[stepIdx]; 	tsv_M18	:= N_RCP_M18[stepIdx];
	tsv_M19	:= N_RCP_M19[stepIdx]; 	
	
	tsv_IH := N_RCP_IH[stepIdx];
	tsv_ROT	:= UINT_TO_REAL(N_RCP_ROT[stepIdx]);
	IF en_TV_posMode THEN
		tsv_POS := N_RCP_POS[stepIdx];	
	ELSE
		tsv_P01 := N_RCP_P01[stepIdx];
	END_IF	
				
	(*Gas valve set*)
	cm_V01 := N_RCP_V01[stepIdx]; cm_V02 := N_RCP_V02[stepIdx];
	cm_V03 := N_RCP_V03[stepIdx]; cm_V04 := N_RCP_V04[stepIdx];
	cm_V05 := N_RCP_V05[stepIdx]; cm_V07 := N_RCP_V07[stepIdx];
	cm_V08 := N_RCP_V08[stepIdx]; cm_V10 := N_RCP_V10[stepIdx];
	cm_V11 := N_RCP_V11[stepIdx]; cm_V13 := N_RCP_V13[stepIdx];
	cm_V14 := N_RCP_V14[stepIdx]; cm_V16 := N_RCP_V16[stepIdx];
	cm_V17 := N_RCP_V17[stepIdx]; cm_V19 := N_RCP_V19[stepIdx];
	cm_V20 := N_RCP_V20[stepIdx]; cm_V22 := N_RCP_V22[stepIdx];
	cm_V23 := N_RCP_V23[stepIdx]; cm_V24 := N_RCP_V24[stepIdx];	
	cm_V25 := N_RCP_V25[stepIdx]; cm_V26 := N_RCP_V26[stepIdx];
	cm_V27 := N_RCP_V27[stepIdx]; cm_V28 := N_RCP_V28[stepIdx];	
	cm_V29 := N_RCP_V29[stepIdx]; cm_V30 := N_RCP_V30[stepIdx];	
	cm_V31 := N_RCP_V31[stepIdx]; cm_V32 := N_RCP_V32[stepIdx];
		
	//Ctemp , Loop. Jump 
	sv_STEP_CTEMP := N_RCP_CTEMP[stepIdx];			
	//Jump & Loop
	IF nLoop = 0 THEN
		sv_STEP_LOOP := N_RCP_LOOP[stepIdx];
		sv_STEP_JUMP := N_RCP_JUMP[stepIdx];
		nLoop := REAL_TO_INT(sv_STEP_LOOP);
		nJump := REAL_TO_INT(sv_STEP_JUMP);										
		IF nLoop > 0 AND nJump > 0 THEN	
			nLoop_Cnt := 0;
			jumpStart := nJump - 1;
			jumpEnd := stepIdx;
		END_IF;
	END_IF;			
	nCase := 20;
END_IF

//Ramping Time || Compare Temp Check
IF nCase = 20 THEN
	//pause
	IF cm_RCP_pause THEN 
		cm_RCP_pause := 0;
		IF s_is_RCP_pause = 0 THEN 
			PT_RAMP_REMAIN := PT_RAMP - ET_RAMP;
			ET_RAMP_RUN := ET_RAMP_RUN + ET_RAMP;
			s_is_RCP_pause := 1; 
		END_IF
	END_IF
	//restart
	IF cm_RCP_restart THEN 
		cm_RCP_restart := 0;
		IF s_is_RCP_pause THEN 
			PT_RAMP := PT_RAMP_REMAIN;
			s_is_RCP_pause := 0;
		END_IF
	END_IF		
	//skip
	IF cm_RCP_skip THEN cm_RCP_skip := 0; T_Ramp(IN:= 0); nCase := 40; END_IF
		
	T_Ramp(IN:= NOT s_is_RCP_pause);
	
	IF 	sv_STEP_CTEMP > 0 THEN//Compare Temp
		//GIST VLC -> FP00_CTemp > 50;
		//Genicom VLC -> FP00_CTemp > 0; 				
		//GIST VLC -> FP00_CTemp -20 < FP00_RTemp_Real   AND   FP00_RTemp_Real < FP00_CTemp + 1;
		//Genicom VLC -> FP00_CTemp -10 < FP00_RTemp_Real   AND   FP00_RTemp_Real < FP00_CTemp + 1;
		//온도를 올릴 때도 있고 내릴 때 비교할 수도 있다.
		//IF IS_RCP_PAUSE = Off AND sv_STEP_CTEMP - 10 < tsv_RTemp AND tsv_RTemp  < sv_STEP_CTEMP + 1  THEN
		IF s_is_RCP_pause = 0 AND sv_STEP_CTEMP - 10 < pv_IH AND pv_IH < sv_STEP_CTEMP + 1 THEN						
			nCase := 40;					
		END_IF				
	ELSE // Normal Ramp			
		IF T_Ramp.Q THEN			
			T_Ramp(IN:= 0);
			nCase := 30;			
		END_IF
	END_IF
		pv_STEP_RTM := F_ET2Sec(IN:= ET_RAMP, SecScale:= SecScale) + F_ET2Sec(IN:= ET_RAMP_RUN, SecScale:= SecScale);	
		pv_RCP_RUN_ET := F_ET2Sec(IN:= ET_RUN, SecScale:= SecScale);
END_IF

//Holding Time
IF nCase = 30 THEN 
	//pause
	IF cm_RCP_pause THEN 
		cm_RCP_pause := 0;
		IF s_is_RCP_pause = 0 THEN 
			PT_HOLD_REMAIN := PT_HOLD - ET_HOLD;
			ET_HOLD_RUN := ET_HOLD_RUN + ET_HOLD;
			s_is_RCP_pause := 1; 
		END_IF
	END_IF
	//restart
	IF cm_RCP_restart THEN 
		cm_RCP_restart := 0;
		IF s_is_RCP_pause THEN 
			PT_HOLD := PT_HOLD_REMAIN;
			s_is_RCP_pause := 0;
		END_IF
	END_IF		
	//skip
	IF cm_RCP_skip  THEN cm_RCP_skip := 0; T_Ramp(IN:= 0); nCase := 40; END_IF	
	//hold time done
	T_Hold(IN:= NOT s_is_RCP_pause);
	IF T_Hold.Q THEN			
		T_Hold(IN:= 0);
		nCase := 40;						
	END_IF
	pv_STEP_HTM := F_ET2Sec(IN:= ET_HOLD, SecScale:= SecScale) + F_ET2Sec(IN:= ET_HOLD_RUN, SecScale:= SecScale);
	pv_RCP_RUN_ET := F_ET2Sec(IN:= ET_RUN, SecScale:= SecScale);
END_IF	

//Loop or Normal Condition Check
IF nCase = 40 THEN
	IF nLoop = 0 THEN
		nCase := 100;
	ELSE
		nCase := 50;
	END_IF;
END_IF

//Loop Next Step Check	
IF nCase = 50 THEN		
	IF stepIdx < jumpEnd THEN 
		stepIdx := stepIdx + 1;
		nCase := 110;
	ELSE						
		IF nLoop <= nLoop_Cnt THEN
			nLoop := 0;
			nLoop_Cnt := 0;
			jumpStart := 0;
			jumpEnd :=	0;
			nCase := 100;
		ELSE
			stepIdx := jumpStart;
			nLoop_Cnt := nLoop_Cnt + 1;	
			nCase := 110;
		END_IF;							 
	END_IF		
END_IF		

//Normal Next Step
IF nCase = 100 THEN
	s_is_RCP_pause := 0;
	stepIdx := stepIdx + 1;
	nCase := 110;
END_IF

//End Checking
IF nCase = 110 THEN
	IF (N_RCP_RTM[stepIdx] = 0 AND N_RCP_HTM[stepIdx]= 0) OR stepIdx >= 200 THEN
		is_RCP_ended := 1;
		s_EN_EXE_RCP := 0;
		nCase := 0;
	ELSE
		T_Ramp(IN:= 0);
		T_Hold(IN:= 0);			
		nCase := 10;
	END_IF
END_IF

IF s_EN_EXE_RCP THEN
	//ramp En Check
	i_RUN_TM := REAL_TO_DINT(pv_RCP_RUN_ET);
	s_P_RampEN := i_RUN_TM_OLD < i_RUN_TM; //Recipe Ramp Call ************************
	i_RUN_TM_OLD := i_RUN_TM;
ELSE // EN_EXE_RCP == 0
	T_Ramp(IN:= 0);
	T_Hold(IN:= 0);
	s_is_RCP_pause := 0;
	s_P_RampEN := 0;
	stepIdx := 0;
	nCase := 0;
END_IF

IF  nCase > 0 AND (is_AL OR is_RCP_ended OR cm_FC_stop) THEN	
	//cm_US1 := On;
	IF is_AL = 0 AND e_US_RCP > 0 THEN
		CASE e_US_RCP OF
			1: cm_US1 := 1;
			2: cm_US2 := 1;
			3: cm_US3 := 1;
			4: cm_US4 := 1;
		END_CASE
	END_IF
		
	pv_STEP_RTM	:= 0;
	pv_STEP_HTM	:= 0;
	pv_RCP_PAUSE_ET	:= 0;
	pv_STEP_LOOP := 0;
	sv_STEP_JUMP := 0;
	s_EN_EXE_RCP := 0;
	//cm_RCP_stop := 0;
	cm_RCP_pause := 0;
	cm_RCP_restart := 0;
	cm_RCP_skip := 0;		
	//cm_ROT_On := 0;
	is_RCP_ended := 0;
	s_is_RCP_pause := 0;
END_IF

pv_RCP_STEP := INT_TO_REAL(stepIdx) + 1;
IF nLoop > 0 AND nJump > 0 THEN
	pv_STEP_JUMP := INT_TO_REAL(jumpStart) + 1;
	pv_STEP_LOOP := INT_TO_REAL(nLoop_Cnt);	
ELSE
	pv_STEP_JUMP := 0;
	pv_STEP_LOOP := 0;
END_IF
ing_RCP_pause := s_is_RCP_pause;
ing_RCP := nCase <> 0;
ing_RCP_ramp := nCase = 20;
ing_RCP_hold := nCase = 30;
ing_RCP_cTemp := ing_RCP_ramp AND sv_STEP_CTEMP > 0;
ing_RCP_loop := nLoop > 0;
pv_RCP_PAUSE_ET := F_ET2Sec(IN:=ET_Pause, SecScale:=SecScale);

END_PROGRAM

// ---- POUs/MR_PRG/P24_Rot_Calibration.TcPOU
PROGRAM P24_Rot_Calibration
VAR
	T1: TON := (PT:= T#1S); //For stabilize //T#500MS
	T2: TON := (PT:= T#1S);; //For Next step//T#200MS
	P_Run: R_TRIG;
	P_Next: R_TRIG;
	Inc_RPM: REAL;
END_VAR

T1(IN:= s_EN_EXE_ROT_CALI);//Timer On
T2(IN:= T1.Q);
P_Run(CLK:= s_EN_EXE_ROT_CALI);
P_Next(CLK:= T2.Q);

IF P_Run.Q THEN
	rtm_ROT := 0;
	tsv_ROT := 0;
	Inc_RPM := 1; //2024-02-20 N_MAX[27] / N_MAX[65]; //Rotation Max RPM / BLDC Max 4000RPM = Inc_RPM
END_IF
	
//Wait until it stabilizes.	
is_ROT_caliStabilized := T1.Q;
is_ROT_caliOn := s_EN_EXE_ROT_CALI;	

//stabil 1sec -> Next
IF P_Next.Q THEN	 
	IF tsv_ROT >= (N_MAX[27]) OR do_ROT = 0 THEN
 		tsv_ROT := 0;
		s_EN_EXE_ROT_CALI := 0;
 	ELSE
		tsv_ROT := tsv_ROT + Inc_RPM;
	 END_IF
	T1(IN:= 0);// Timer Reset
END_IF

END_PROGRAM

// ---- POUs/MR_PRG/P25_US_Ctrl.TcPOU
PROGRAM P25_US_Ctrl
VAR
	i: INT;
	idx: INT;
	rampSteps: REAL;
END_VAR

//idx := REAL_TO_INT(tsv_US);

idx := -1;
IF cm_US1 THEN
	idx := 0;
ELSIF cm_US2 THEN
	idx := 1;
ELSIF cm_US3 THEN
	idx := 2;
ELSIF cm_US4 THEN
	idx := 3;
END_IF


//Maint Mode에서 User State 금지
IF ing_MAINT AND -1 < idx THEN
	idx := -1;
END_IF

IF 0 <= idx AND idx<= 3 THEN
	
	rampSteps := N_US_A[idx, 0];
	IF rampSteps < 1 THEN rampsteps := 1; END_IF;
	
	//Analog Set
	//genicom - M01 ~ M19, E01~E07, RTEMP, PRES까지 , ROT 제외
	FOR i := 0 TO 29 DO	
		//TSV Set
		N_TSV_RTM[i * 2] := N_US_A[idx, i + 1];	
         //RTM Set	
		IF N_EN_RAMP[i]THEN	
			N_TSV_RTM[i * 2 + 1] := rampsteps;
		ELSE
			N_TSV_RTM[i * 2 + 1] := 0;	
		END_IF				   			
	END_FOR  
	
	IF is_TCAT_started = 0 THEN
		sv_P01 := tsv_P01;
		rtm_P01 := 0;
	END_IF
		
	IF N_US_D[idx, 0] = 1 THEN cm_V01 := 1; ELSIF  N_US_D[idx, 0] = 2 THEN  cm_V01 := 0; END_IF
	IF N_US_D[idx, 1] = 1 THEN cm_V02 := 1; ELSIF  N_US_D[idx, 1] = 2 THEN  cm_V02 := 0; END_IF
	IF N_US_D[idx, 2] = 1 THEN cm_V03 := 1; ELSIF  N_US_D[idx, 2] = 2 THEN  cm_V03 := 0; END_IF	
	IF N_US_D[idx, 3] = 1 THEN cm_V04 := 1; ELSIF  N_US_D[idx, 3] = 2 THEN  cm_V04 := 0; END_IF
	IF N_US_D[idx, 4] = 1 THEN cm_V05 := 0; ELSIF  N_US_D[idx, 4] = 2 THEN  cm_V05 := 1; END_IF //N.O Valve	
	IF N_US_D[idx, 5] = 1 THEN cm_V07 := 1; ELSIF  N_US_D[idx, 5] = 2 THEN  cm_V07 := 0; END_IF	
	IF N_US_D[idx, 6] = 1 THEN cm_V08 := 0; ELSIF  N_US_D[idx, 6] = 2 THEN  cm_V08 := 1; END_IF //N.O Valve
	IF N_US_D[idx, 7] = 1 THEN cm_V10 := 1; ELSIF  N_US_D[idx, 7] = 2 THEN  cm_V10 := 0; END_IF
	IF N_US_D[idx, 8] = 1 THEN cm_V11 := 0; ELSIF  N_US_D[idx, 8] = 2 THEN  cm_V11 := 1; END_IF //N.O Valve
	IF N_US_D[idx, 9] = 1 THEN cm_V13 := 1; ELSIF  N_US_D[idx, 9] = 2 THEN  cm_V13 := 0; END_IF
	IF N_US_D[idx, 10] = 1 THEN cm_V14 := 0; ELSIF  N_US_D[idx, 10] = 2 THEN  cm_V14 := 1; END_IF //N.O Valve
	IF N_US_D[idx, 11] = 1 THEN cm_V16 := 1; ELSIF  N_US_D[idx, 11] = 2 THEN  cm_V16 := 0; END_IF
	IF N_US_D[idx, 12] = 1 THEN cm_V17 := 0; ELSIF  N_US_D[idx, 12] = 2 THEN  cm_V17 := 1; END_IF //N.O Valve
	IF N_US_D[idx, 13] = 1 THEN cm_V19 := 1; ELSIF  N_US_D[idx, 13] = 2 THEN  cm_V19 := 0; END_IF
	IF N_US_D[idx, 14] = 1 THEN cm_V20 := 0; ELSIF  N_US_D[idx, 14] = 2 THEN  cm_V20 := 1; END_IF //N.O Valve
	IF N_US_D[idx, 15] = 1 THEN cm_V22 := 1; ELSIF  N_US_D[idx, 15] = 2 THEN  cm_V22 := 0; END_IF
	IF N_US_D[idx, 16] = 1 THEN cm_V23 := 1; ELSIF  N_US_D[idx, 16] = 2 THEN  cm_V23 := 0; END_IF		
	IF N_US_D[idx, 17] = 1 THEN cm_V24 := 1; ELSIF  N_US_D[idx, 17] = 2 THEN  cm_V24 := 0; END_IF		
	IF N_US_D[idx, 18] = 1 THEN cm_V25 := 1; ELSIF  N_US_D[idx, 18] = 2 THEN  cm_V25 := 0; END_IF
	IF N_US_D[idx, 19] = 1 THEN cm_V26 := 1; ELSIF  N_US_D[idx, 19] = 2 THEN  cm_V26 := 0; END_IF		
	IF N_US_D[idx, 20] = 1 THEN cm_V27 := 1; ELSIF  N_US_D[idx, 20] = 2 THEN  cm_V27 := 0; END_IF		
	IF N_US_D[idx, 21] = 1 THEN cm_V28 := 1; ELSIF  N_US_D[idx, 21] = 2 THEN  cm_V28 := 0; END_IF		
	IF N_US_D[idx, 22] = 1 THEN cm_V29 := 1; ELSIF  N_US_D[idx, 22] = 2 THEN  cm_V29 := 0; END_IF				
	IF N_US_D[idx, 23] = 1 THEN cm_V30 := 1; ELSIF  N_US_D[idx, 23] = 2 THEN  cm_V30 := 0; END_IF
	IF N_US_D[idx, 24] = 1 THEN cm_V31 := 1; ELSIF  N_US_D[idx, 24] = 2 THEN  cm_V31 := 0; END_IF
	IF N_US_D[idx, 25] = 1 THEN cm_V32 := 1; ELSIF  N_US_D[idx, 25] = 2 THEN  cm_V32 := 0; END_IF	
			
	//TV------------------------------Check
	IF N_US_D[idx, 26] > 0 THEN		
		IF N_US_D[idx, 26] = 1 THEN//Run[Torr]
			en_TV_posMode := 0;
			cm_TV_Run := 1;
		ELSIF  N_US_D[idx, 26] = 2 THEN//Run[%]
			en_TV_posMode := 1;
			cm_TV_Run := 1;
		ELSIF  N_US_D[idx, 26] = 3 THEN//Open    	
			cm_TV_open := 1;
		ELSIF  N_US_D[idx, 26] = 4 THEN//Close    	
			cm_TV_close := 1;
		ELSIF  N_US_D[idx, 26] = 5 THEN//Hold == Stop    	
			cm_TV_stop := 1;
		END_IF
	END_IF

	//tsv_ROT := 0;
	//rtm_ROT := rampsteps;

    pv_US := idx;
END_IF;

cm_US1 := cm_US2 := cm_US3 := cm_US4 := 0;

(*
IF idx2 > -1 THEN
	IF 	tsv_M00 = N_US_A[idx2, 1]  AND
		tsv_M01 = N_US_A[idx2, 2]  AND
		tsv_M02 = N_US_A[idx2, 3]  AND
		tsv_M03 = N_US_A[idx2, 4]  AND
		tsv_M04 = N_US_A[idx2, 5]  AND
		tsv_M05 = N_US_A[idx2, 6]  AND
		tsv_M06 = N_US_A[idx2, 7]  AND
		tsv_M07 = N_US_A[idx2, 8]  AND
		tsv_M08 = N_US_A[idx2, 9]  AND
		tsv_M09 = N_US_A[idx2, 10]  AND
		tsv_M10 = N_US_A[idx2, 11]  AND
		tsv_M11 = N_US_A[idx2, 12]  AND
		tsv_M12 = N_US_A[idx2, 13]  AND
		tsv_M13 = N_US_A[idx2, 14]  AND
		tsv_M14 = N_US_A[idx2, 15]  AND
		tsv_M15 = N_US_A[idx2, 16]  AND
		tsv_M16 = N_US_A[idx2, 17]  AND
		tsv_M17 = N_US_A[idx2, 18]  AND
		tsv_M18 = N_US_A[idx2, 19]  AND
		tsv_M19 = N_US_A[idx2, 20]  AND
		tsv_M20 = N_US_A[idx2, 21]  AND
		tsv_E01 = N_US_A[idx2, 22]  AND
		tsv_E02 = N_US_A[idx2, 23]  AND
		tsv_E03 = N_US_A[idx2, 24]  AND
		tsv_E04 = N_US_A[idx2, 25]  AND
		tsv_E05 = N_US_A[idx2, 26]  AND
		tsv_E06 = N_US_A[idx2, 27]  AND
		tsv_RTEMP = N_US_A[idx2, 28]  AND
		tsv_PRES = N_US_A[idx2, 29]  AND
		
		cm_V00 = N_US_D[idx2, 0]  AND
		cm_V01 = N_US_D[idx2, 1]  AND
		cm_V02 = N_US_D[idx2, 2]  AND
		cm_V03 = N_US_D[idx2, 3]  AND
		cm_V04 = N_US_D[idx2, 4]  AND
		cm_V05 = N_US_D[idx2, 5]  AND
		cm_V06 = N_US_D[idx2, 6]  AND
		cm_V07 = N_US_D[idx2, 7]  AND
		cm_V08 = N_US_D[idx2, 8]  AND
		cm_V09 = N_US_D[idx2, 9]  AND
		cm_V10 = N_US_D[idx2, 10]  AND
		cm_V11 = N_US_D[idx2, 11]  AND
		cm_V12 = N_US_D[idx2, 12]  AND
		cm_V13 = N_US_D[idx2, 13]  AND
		cm_V14 = N_US_D[idx2, 14]  AND
		cm_V15 = N_US_D[idx2, 15]  AND
		cm_V16 = N_US_D[idx2, 16]  AND
		cm_V17 = N_US_D[idx2, 17]  AND
		cm_V18 = N_US_D[idx2, 18]  AND
		cm_V19 = N_US_D[idx2, 19]  AND
		cm_V20 = N_US_D[idx2, 20]  AND
		cm_V21 = N_US_D[idx2, 21]  AND
		cm_V22 = N_US_D[idx2, 22]  AND
		cm_V24 = N_US_D[idx2, 23]  AND
		cm_V25 = N_US_D[idx2, 24]  AND
		cm_V26 = N_US_D[idx2, 25]  THEN
		pv_US := idx2;
	ELSE
		pv_US := -1;
	END_IF;

END_IF;
*)

END_PROGRAM

// ---- POUs/MR_PRG/P31_BypassV.TcPOU
PROGRAM P31_BypassV
VAR
	p_OverP_UP: R_TRIG;
	p_OverP_DW: F_TRIG;
END_VAR


//Over Pressure Bypass Valve
//VLC에서 V26 On/Off 제어 로직이 없음
IF ing_MAINT THEN
	p_OverP_UP(CLK:= is_TV_close AND is_P01_overP_al);
	p_OverP_DW(CLK:= is_P01_overP_al);
	IF p_OverP_UP.Q THEN
		cm_V33_1 := 0;
		cm_V33_2 := 0;
	END_IF
	IF p_OverP_DW.Q THEN
		cm_V33_1 := 0;
		cm_V33_2 := 1;
	END_IF	
ELSE
	IF is_TV_close THEN
		cm_V33_1 := cm_V33_2 := is_P01_overP_al = 1;
	ELSE
		cm_V33_1 := 0;
		cm_V33_2 := 1;
	END_IF
END_IF;

END_PROGRAM

// ---- POUs/MR_PRG/P41_DOR_VAC.TcPOU
PROGRAM P41_DOR_VAC
VAR
	p_Start, p_EMS: R_TRIG;
	nCase: INT;
	T1: TON;
	PT1: TIME := T#1S;
	T_Blink: TON := (PT:= T#1S);
END_VAR

//DOR 진공 잡기
//is_DOR_05Bar : 약 375Torr
//is_DOR_01Bar : 약 75Torr

T1(IN:= s_EN_EXE_DOR_VAC, PT:= PT1);
T_Blink(IN:= nCase > 0);
p_Start(CLK:= s_EN_EXE_DOR_VAC);
p_EMS(CLK:= (nCase > 0 AND s_EN_EXE_DOR_VAC = 0) OR is_AL);

IF p_Start.Q THEN
	nCase := 1;
END_IF

IF p_EMS.Q THEN
	s_EN_EXE_DOR_VAC := 0;
	nCase := 0;
END_IF


CASE nCase OF
	1://Init
		is_DOR_ATM_ok := 0;
		en_SH_UpDw := 0;
		s_DOR_CNT := 0;
		cm_V35 := 0;//DOR Vent
		cm_V34 := 1;//DOR Vacuum
		PT1 := T#2S;
		T1(IN:= 0);
		nCase := 2;
	2://1st wait
		IF T1.Q THEN
			T1(IN:= 0);
			nCase := 10;
		END_IF
	10://1st vac check
		IF T1.Q THEN//2sec pulse
			T1(IN:= 0);
			IF is_DOR_05ATM AND is_DOR_01ATM THEN
				s_DOR_CNT := 0;
				nCase := 20;
			ELSE
				s_DOR_CNT := s_DOR_CNT + 1;//1st DOR AL&WN Check
			END_IF
		END_IF
	20://2st vac check 
		IF T1.Q THEN//2sec pulse
			T1(IN:= 0);
			IF is_DOR_05ATM AND is_DOR_01ATM THEN				
				cm_V34 := e_d_V34_keep_on;//DOR VAC				
				cm_V35 := 0;//DOR ATM				
				is_DOR_VAC_ok := 1;
				s_EN_EXE_DOR_VAC := 0;
				nCase := 0;
			ELSE
				s_DOR_CNT := s_DOR_CNT + 1;//2st DOR AL&WN Check
			END_IF
		END_IF
END_CASE


IF s_EN_EXE_DOR_VAC THEN
	IF T_Blink.Q THEN
		T_Blink(IN := 0);
		is_DOR_VAC_blink := NOT is_DOR_VAC_blink;
	END_IF
ELSE
	is_DOR_VAC_blink := 0;
END_IF;

END_PROGRAM

// ---- POUs/MR_PRG/P41_DOR_VAC_Check.TcPOU
PROGRAM P41_DOR_VAC_Check
VAR
	T1: TON := (PT:= T#10S);
	re_DOR_ok: BOOL;
END_VAR

//DOR 진공이 is_DOR_05Bar 이상 깨지면 다시 진공 잡기
//is_DOR_05Bar : 약 375Torr
//is_DOR_01Bar : 약 75Torr

//GIST VLC Manual_SH_Vacum_Check
//Genicom VLC Manual_SH_Vacum_Check

IF is_DOR_VAC_ok AND di_VP_busy THEN	
	IF is_DOR_05ATM = 0 THEN//진공이 떨어지면 자동 밸브 작동 		
		T1(IN:= 1);		
		s_is_DOR_Broken := 0;	
		re_DOR_ok := 0;
		cm_V34 := 1;//DOR VAC
		cm_V35 := 0;//DOR ATM			
	END_IF
	
	IF T1.Q THEN // Dor Check
		T1(IN:= 0);
		IF is_DOR_05ATM AND is_DOR_01ATM THEN // Dor Check
			re_DOR_ok := 1;
		ELSE
			s_is_DOR_Broken := 1;		
		END_IF;
	END_IF
	
	IF re_DOR_ok THEN // Dor End
		re_DOR_ok := 0;
		cm_V34 := e_d_V34_keep_on;//DOR VAC				
		cm_V35 := 0;//DOR ATM	
	END_IF
END_IF

END_PROGRAM

// ---- POUs/MR_PRG/P42_DOR_ATM.TcPOU
PROGRAM P42_DOR_ATM
VAR
	p_Start, p_EMS: R_TRIG;
	T1: TON;
	PT1: TIME := T#1S;
	ET1: TIME;
	T_Blink: TON := (PT:= T#1S);
	rampSec: REAL;
	nCase: INT;
END_VAR

//VLC Manual_SH_Up.flo
T1(PT:= PT1, ET=> ET1);
T_Blink(IN:= nCase > 0);
p_Start(CLK:= s_EN_EXE_DOR_ATM);
p_EMS(CLK:= (nCase > 0 AND s_EN_EXE_DOR_ATM = 0) OR is_AL);

IF p_Start.Q THEN
	nCase := 1;
END_IF

IF p_EMS.Q THEN
	s_EN_EXE_DOR_ATM := 0;
	nCase := 0;
END_IF

en_DOR_ATM := ing_RCP = 0 AND
				 is_AL = 0 AND
				 pv_IH <= e_EN_DOR_ATM_IH  AND
				 pv_P01 >= e_EN_DOR_ATM_P01 AND
				 do_V01 = 0 AND // H2 Supply
				 do_V02 = 0 AND // H2 Supply				 
				 do_V03 = 0 AND //SiH4 Supply
				 do_V04 = 0 AND //NH3 Supply
				 di_SH_lo_limit; 
				 
CASE nCase OF
	1://US Set
		is_DOR_VAC_ok := is_DOR_ATM_ok := 0;
		en_SH_UpDw := 0;
		rampSec := 1;	
		IF e_US_DOR_ATM > 0 THEN
			CASE e_US_DOR_ATM OF
				1: 
					cm_US1 := 1;
					rampSec := N_US_A[0,0];//US1 RampStep
				2: 
					cm_US2 := 1;
					rampSec := N_US_A[1,0];//US2 RampStep
				3: 
					cm_US3 := 1;
					rampSec := N_US_A[2,0];//US3 RampStep
				4: 
					cm_US4 := 1;
					rampSec := N_US_A[3,0];//US4 RampStep
			END_CASE
		END_IF

		IF rampSec <= 0 THEN rampSec := 10; END_IF//Default 10Sec							
		rampSec := rampSec * 2;//램프시간의 2배를 기다린다.		
		pv_DOR_ATM_cnt := rampSec;		
		PT1 := REAL_TO_TIME(rampSec * 1000);
		T1(IN:= 1);			
		nCase := 2;
	2:
		IF T1.Q THEN
			T1(IN:= 0);	
			cm_V34 := 0;//DOR VAC
			cm_V35 := 1;//DOR ATM			
			nCase := 10;
		END_IF
	10://Wait
		PT1 := T#2S;
		T1(IN:= 1);		
		nCase := 11;
	11:
		IF T1.Q THEN
			T1(IN:= 0);
			nCase := 20;
		END_IF					
	20: //Open Codition Check
		IF pv_P01 >= e_EN_DOR_ATM_P01 AND pv_IH <= e_EN_DOR_ATM_IH //PRES > 750 && RTEMP < 500
			AND is_DOR_1ATM THEN
			nCase := 0; //FC Stop
			cm_V35 := 0;//DOR ATM
			is_DOR_ATM_ok := 1;
			en_SH_UpDw := 1;
		ELSE
			nCase := 0; //FC Stop
		END_IF	
		s_EN_EXE_DOR_ATM := 0;
END_CASE


//IF en_SH_UpDw = 0 THEN
	//is_DOR_ATM_blink := 0;
//END_IF

IF T_Blink.Q THEN
	T_Blink(IN:= 0);
	pv_DOR_ATM_cnt := pv_DOR_ATM_cnt - 1;
	IF pv_DOR_ATM_cnt < 0 THEN pv_DOR_ATM_cnt := 0; END_IF;
	is_DOR_ATM_blink := NOT is_DOR_ATM_blink;
ELSIF nCase <= 0 THEN
	is_DOR_ATM_blink := 0;
END_IF

END_PROGRAM

// ---- POUs/MR_PRG/P43_SH_UpDw.TcPOU
PROGRAM P43_SH_UpDw
VAR	
	//For Led Display
	T_UP: TON := (PT:= T#200MS);
	T_UP_X: TON := (PT:= T#200MS);
	T_DW: TON := (PT:= T#200MS);
	T_DW_X: TON := (PT:= T#200MS);
	//For S/H Down Delay
	T_DW_off: TON := (PT:= T#1S);
END_VAR

T_UP(IN:= do_SH_up_ry AND T_UP_X.Q = 0);
T_UP_X(IN:= T_UP.Q);

T_DW(IN:= do_SH_dw_ry AND T_DW_X.Q = 0);
T_DW_X(IN:= T_DW.Q);

//en_SH_UpDw:= 1;//TEST
T_DW_off(IN:= di_SH_lo_limit);
IF en_SH_UpDw THEN
   cm_SH_up_ry := di_SH_dw = 0 AND di_SH_up AND di_SH_hi_limit = 0;
   cm_SH_dw_ry := di_SH_up = 0 AND di_SH_dw AND (di_SH_lo_limit = 0 OR T_DW_off.Q = 0);
END_IF


cm_SH_up_led := (T_UP.Q = 0 AND cm_SH_up_ry) OR di_SH_hi_limit;
cm_SH_dw_led := (T_DW.Q = 0 AND cm_SH_dw_ry) OR di_SH_lo_limit;

END_PROGRAM

// ---- POUs/MR_PRG/P49_MO_SRC.TcPOU
PROGRAM P49_MO_SRC
VAR
	_1mole_volume: REAL := 22400;//1몰 부피 = 1/22400
	//_1mole_volume: REAL := 0.0000000744047619;//1.0/22400.0/60.0;//1몰 부피 = 1/22400 * 1/60 미리 계산
	
	T_1S: TON := (PT:= T#1S);
	
	T1: TON := (PT:= T#1S);
	ms1_K, ms1_data1, ms1_data2: REAL;
	
	T2: TON := (PT:= T#1S);
	ms2_K, ms2_data1, ms2_data2: REAL;
	
	T3: TON := (PT:= T#1S);
	ms3_K, ms3_data1, ms3_data2: REAL;
	
	T4: TON := (PT:= T#1S);
	ms4_K, ms4_data1, ms4_data2: REAL;
	
	T5: TON := (PT:= T#1S);
	ms5_K, ms5_data1, ms5_data2: REAL;
	
	T6: TON := (PT:= T#1S);
	ms6_K, ms6_data1, ms6_data2: REAL;
	ms6_ln: REAL;
	
(*	//Old
	t0 : TON;
	ms0_Vapor : REAL := 1; //설정
	ms0_Bub_Const : REAL :=1; //설정
	ms0_data1 : REAL;
	ms0_data2 : REAL;
	ms0_data3 : REAL;
	ms0_inc : REAL;
	m00_csv : REAL;
	
	t1 : TON;
	ms1_Vapor : REAL := 1; //설정
	ms1_Bub_Const : REAL :=1; //설정
	ms1_data1 : REAL;
	ms1_data2 : REAL;
	ms1_data3 : REAL;
	ms1_inc : REAL;
	m01_csv : REAL;
	
	t2 : TON;
	ms2_Vapor : REAL := 1; //설정
	ms2_Bub_Const : REAL :=1; //설정
	ms2_data1 : REAL;
	ms2_data2 : REAL;
	ms2_data3 : REAL;
	ms2_inc : REAL;
	m02_csv : REAL;
	
	t3 : TON;
	ms3_Vapor : REAL := 1; //설정
	ms3_Bub_Const : REAL :=1; //설정
	ms3_data1 : REAL;
	ms3_data2 : REAL;
	ms3_data3 : REAL;
	ms3_inc : REAL;
	m03_csv : REAL;
	
	t4 : TON;
	ms4_Vapor : REAL := 1; //설정
	ms4_Bub_Const : REAL :=1; //설정
	ms4_data1 : REAL;
	ms4_data2 : REAL;
	ms4_data3 : REAL;
	ms4_inc : REAL;
	m04_csv : REAL;
*)	
	
END_VAR

T_1S(IN := 1);
IF T_1S.Q THEN
	T_1S(IN := 0);
	
	//MO1 - TEB : 부분압 구하기  pow(10, (a - ( b / T )))	
	IF N_MS_SET[0, 0] < 1 THEN// 상수 온도 사용
		ms1_K := N_MS_SET[0, 3] + 273.16; //절대 온도로 변환
	ELSE //측정 온도 사용
		ms1_K := pv_TB1 + 273.16; //절대 온도로 변환	
	END_IF	
	pv_MS1_Pres := EXPT(10, (N_MS_SET[0, 1] - ( N_MS_SET[0, 2] / ms1_K)));
	
	//MO2 - TMAI : 부분압 구하기  pow(10, (a - ( b / T )))	
	IF N_MS_SET[1, 0] < 1 THEN// 상수 온도 사용
		ms2_K := N_MS_SET[1, 3] + 273.16; //절대 온도로 변환
	ELSE //측정 온도 사용
		ms2_K := pv_TB2 + 273.16; //절대 온도로 변환	
	END_IF	
	pv_MS2_Pres := EXPT(10, (N_MS_SET[1, 1] - ( N_MS_SET[1, 2] / ms2_K)));
	
	//MO3 - TMIn : 부분압 구하기  pow(10, (a - ( b / T )))
	IF N_MS_SET[2, 0] < 1 THEN// 상수 온도 사용
		ms3_K := N_MS_SET[2, 3] + 273.16; //절대 온도로 변환
	ELSE //측정 온도 사용
		ms3_K := pv_TB3 + 273.16; //절대 온도로 변환	
	END_IF	
	pv_MS3_Pres := EXPT(10, (N_MS_SET[2, 1] - ( N_MS_SET[2, 2] / ms3_K)));
	
	//MO4 - TMGa : 부분압 구하기  pow(10, (a - ( b / T )))	
	IF N_MS_SET[3, 0] < 1 THEN// 상수 온도 사용
		ms4_K := N_MS_SET[3, 3] + 273.16; //절대 온도로 변환
	ELSE //측정 온도 사용
		ms4_K := pv_TB4 + 273.16; //절대 온도로 변환	
	END_IF	
	pv_MS4_Pres := EXPT(10, (N_MS_SET[3, 1] - ( N_MS_SET[3, 2] / ms4_K)));
	
	//MO5 - DTMGa : 부분압 구하기  pow(10, (a - ( b / T )))
	IF N_MS_SET[4, 0] < 1 THEN// 상수 온도 사용
		ms5_K := N_MS_SET[4, 3] + 273.16; //절대 온도로 변환
	ELSE //측정 온도 사용
		ms5_K := pv_TB5 + 273.16; //절대 온도로 변환	
	END_IF	
	pv_MS5_Pres := EXPT(10, (N_MS_SET[4, 1] - ( N_MS_SET[4, 2] / ms5_K)));
	

	//MO6 - Cp2Mg(고체) : 부분압 구하기  pow(10, (a - 2.18LN(T) - ( b / T )))
	IF N_MS_SET[5, 0] < 1 THEN// 상수 온도 사용
		ms6_K := N_MS_SET[5, 3] + 273.16; //절대 온도로 변환
	ELSE //측정 온도 사용
		ms6_K := pv_TB6 + 273.16; //절대 온도로 변환	
	END_IF	
	//LN()
	//The IEC operator returns the natural logarithm OF a number.
    //Permitted data types for the input variables: any numeric basic data type
    //Permitted data types for the output variables: REAL and LREAL
	ms6_ln := 2.18 * LN(ms6_K);	
	pv_MS6_Pres := EXPT(10, (N_MS_SET[5, 1] - ms6_ln - ( N_MS_SET[5, 2] / ms6_K))); //
		
END_IF


//Mo 소스 무게 계산 
//MO1 - TEB
T1(IN:= do_V07);
IF T1.Q THEN
	T1(IN:= 0);	
	IF pv_E02 > 10 AND pv_M08 > 0 AND pv_MS1_Pres > 0 THEN				
		ms1_data1 := pv_M08 * (pv_MS1_Pres / (pv_E02 - pv_MS1_Pres)) / _1mole_volume / 60; //formular2-1		
		ms1_data2 := ms1_data1 * N_MS_SET[0, 4] * N_MS_SET[0, 5]; //formular2-2		
		N_MS_SET[0, 7] := N_MS_SET[0, 7] + ms1_data2; //used Weight
	END_IF	
END_IF
pv_MS1 := N_MS_SET[0, 8] := N_MS_SET[0, 6] - N_MS_SET[0, 7]; //remain Weight


//MO2 - TMAI
T2(IN:= do_V10);
IF T2.Q THEN
	T2(IN:= 0);
	IF pv_E03 > 10 AND pv_M09 > 0 AND pv_MS2_Pres > 0 THEN				
		ms2_data1 := pv_M09 * (pv_MS2_Pres / (pv_E03 - pv_MS2_Pres)) / _1mole_volume / 60; //formular2-1		
		ms2_data2 := ms2_data1 * N_MS_SET[1, 4] * N_MS_SET[1, 5]; //formular2-2		
		N_MS_SET[1, 7] := N_MS_SET[1, 7] + ms2_data2; //used Weight
	END_IF
END_IF
pv_MS2 := N_MS_SET[1, 8] := N_MS_SET[1, 6] - N_MS_SET[1, 7]; //remain Weight


//MO3 - TMIn
T3(IN:= do_V13);
IF T3.Q THEN
	T3(IN:= 0);
	IF pv_E04 > 10 AND pv_M10 > 0 AND pv_MS3_Pres > 0 THEN		
		ms3_data1 := pv_M10 * (pv_MS3_Pres / (pv_E04 - pv_MS3_Pres)) / _1mole_volume / 60; //formular2-1	
		ms3_data2 := ms3_data1 * N_MS_SET[2, 4] * N_MS_SET[2, 5]; //formular2-2		
		N_MS_SET[2, 7] := N_MS_SET[2, 7] + ms3_data2; //used Weight
	END_IF	
END_IF
pv_MS3 := N_MS_SET[2, 8] := N_MS_SET[2, 6] - N_MS_SET[2, 7]; //remain Weight


//MO4 - TMGa
T4(IN:= do_V16);
IF T4.Q THEN
	T4(IN:= 0);
	IF pv_E05 > 10 AND pv_M11 > 0 AND pv_MS4_Pres > 0 THEN			
		ms4_data1 := pv_M11 * (pv_MS4_Pres / (pv_E05 - pv_MS4_Pres)) / _1mole_volume / 60; //formular2-1		
		ms4_data2 := ms4_data1 * N_MS_SET[3, 4] * N_MS_SET[3, 5]; //formular2-2		
		N_MS_SET[3, 7] := N_MS_SET[3, 7] + ms4_data2; //used Weight
	END_IF		
END_IF
pv_MS4 := N_MS_SET[3, 8] := N_MS_SET[3, 6] - N_MS_SET[3, 7]; //remain Weight


//MO5 - DTMGa -- MFC is 2 More -> Check Formula -> M12 ok
T5(IN := do_V19);
IF T5.Q THEN
	T5(IN:= 0);
	IF pv_E06 > 10 AND pv_M12 > 0 AND pv_MS5_Pres > 0 THEN			
		ms5_data1 := pv_M12 * (pv_MS5_Pres / (pv_E06 - pv_MS5_Pres)) / _1mole_volume / 60; //formular2-1		
		ms5_data2 := ms5_data1 * N_MS_SET[4, 4] * N_MS_SET[4, 5]; //formular2-2		
		N_MS_SET[4, 7] := N_MS_SET[4, 7] + ms5_data2; //used Weight
	END_IF		
END_IF
pv_MS5 := N_MS_SET[4, 8] := N_MS_SET[4, 6] - N_MS_SET[4, 7]; //remain Weight


//MO6 Cp2Mg
T6(IN := do_V22);
IF T6.Q THEN
	T6(IN:= 0);
	IF pv_E07 > 10 AND pv_M15 > 0 AND pv_MS6_Pres > 0 THEN				
		ms6_data1 := pv_M15 * (pv_MS6_Pres / (pv_E07 - pv_MS6_Pres)) / _1mole_volume / 60; //formular2-1		
		ms6_data2 := ms6_data1 * N_MS_SET[5, 4] * N_MS_SET[5, 5]; //formular2-2	
		N_MS_SET[5, 7] := N_MS_SET[5, 7] + ms6_data2; //used Weight
	END_IF		
END_IF
pv_MS6 := N_MS_SET[5, 8] := N_MS_SET[5, 6] - N_MS_SET[5, 7]; //remain Weight




(* //Old Version
//Mo 소스 무게 계산 -> 제니컴 모드
//TMAI
t0(PT := T#1S);
t0.IN := DO_V01;

IF DO_V01 THEN
	m00_csv := tsv_M00;
	ms0_inc := 0;
END_IF

IF t0.Q THEN
	t0.IN := Off;
	ms0_inc := ms0_inc + 1;	
	IF tsv_E01 > 10 THEN
		//ms0_data1 = 8.224 -  2134.83 / (273 + MO_TMAI_Temp)
		ms0_data1 := ms1_Vapor * tsv_M00/tsv_E01;
		ms0_data2 := ms0_inc * 0.001;
		ms0_data3 := 72.10/1.344;
		pv_MO_SRC1 := pv_MO_SRC1 - ms0_data1 * ms0_data2  * ms0_data3 * ms0_Bub_Const * 0.001;
	END_IF
END_IF


//TMIn
t1(PT := T#1S);
t1.IN := DO_V04;

IF DO_V04 THEN
	m01_csv := tsv_M01;
	ms1_inc := 0;
END_IF

IF t1.Q THEN
	t1.IN := Off;
	ms1_inc := ms1_inc + 1;	
	IF tsv_E02 > 10 THEN
		ms1_data1 := ms1_Vapor * tsv_M01/tsv_E02;
		ms1_data2 := ms1_inc * 0.001;
		ms1_data3 := 159.93/1.344;
		pv_MO_SRC2 := pv_MO_SRC2 - ms1_data1 * ms1_data2  * ms1_data3 * ms1_Bub_Const * 0.001;
	END_IF
END_IF


//TMGa1
t2(PT := T#1S);
t2.IN := DO_V07;

IF DO_V07 THEN
	m02_csv := tsv_M02;
	ms2_inc := 0;
END_IF

IF t2.Q THEN
	t2.IN := Off;
	ms2_inc := ms2_inc + 1;	
	IF tsv_E03 > 10 THEN
		ms2_data1 := ms2_Vapor * tsv_M02/tsv_E03;
		ms2_data2 := ms2_inc * 0.001;
		ms2_data3 := 114.83/1.344;
		pv_MO_SRC3 := pv_MO_SRC3 - ms2_data1 * ms2_data2  * ms2_data3 * ms2_Bub_Const * 0.001;
	END_IF
END_IF


//TMGa2
t3(PT := T#1S);
t3.IN := DO_V10;

IF DO_V10 THEN
	m03_csv := tsv_M03;
	ms3_inc := 0;
END_IF

IF t3.Q THEN
	t3.IN := Off;
	ms3_inc := ms3_inc + 1;	
	IF tsv_E04 > 10 THEN
		//ms3_data1 = 8.07 -  1703 / (273 + MO_TMGa2_Temp)
		ms3_data1 := ms3_Vapor * tsv_M03/tsv_E04;
		ms3_data2 := ms3_inc * 0.001;
		ms3_data3 := 114.83/1.344;
		pv_MO_SRC4 := pv_MO_SRC4 - ms3_data1 * ms3_data2  * ms3_data3 * ms3_Bub_Const * 0.001;
	END_IF
END_IF


//Cp2Mg
t4(PT := T#1S);
t4.IN := DO_V13;

IF DO_V13 THEN
	m04_csv := tsv_M06;
	ms4_inc := 0;
END_IF

IF t4.Q THEN
	t4.IN := Off;
	ms4_inc := ms4_inc + 1;	
	IF tsv_E05 > 10 THEN
		//ms4_data1 = 10.452 -  3522 / (273 + MO_Cp2Mg_Temp)
		ms4_data1 := ms4_Vapor * tsv_M06/tsv_E05;
		ms4_data2 := ms4_inc * 0.001;
		ms4_data3 := 154.49/1.344;
		pv_MO_SRC5 := pv_MO_SRC5 - ms4_data1 * ms4_data2  * ms4_data3 * ms4_Bub_Const * 0.001;
	END_IF
END_IF
*)

END_PROGRAM

// ---- POUs/MR_PRG/P62_Tx_TV.TcPOU
PROGRAM P62_Tx_TV
VAR
	p_TV_RST: R_TRIG;
	Resolution: REAL := 32767;//0~7FFF	
END_VAR

//Throttle Valve - Mode
IF cm_TV_run THEN
	 Tx_TV_Mode := 0;
	 cm_TV_run := 0;
END_IF;
IF cm_TV_close THEN
	 Tx_TV_Mode := 1;
	 cm_TV_close := 0;
END_IF;
IF cm_TV_open THEN
	 Tx_TV_Mode := 2;
	 cm_TV_open := 0;
END_IF;
IF cm_TV_stop THEN
	 Tx_TV_Mode := 3;
	 cm_TV_stop := 0;
END_IF;

//Throttle Valve - Reset
p_TV_RST(CLK:= s_cm_RST AND is_TV_fail);
IF p_TV_RST.Q THEN
	 Tx_TV_Mode := 4;
END_IF;

//Throttle Valve - Set Point
IF en_TV_posMode THEN
	Tx_TV_SP_Type := 2;//positon
	Tx_TV_SP := REAL_TO_WORD(sv_POS * Resolution / N_MAX[28]);//TV POS	
ELSE
	Tx_TV_SP_Type := 1;//pressure
	Tx_TV_SP := REAL_TO_WORD(sv_P01 * Resolution / N_MAX[29]);//P01	
END_IF

END_PROGRAM

// ---- POUs/MR_PRG/P63_Tx_IH.TcPOU
PROGRAM P63_Tx_IH
VAR
	r1: REAL;
END_VAR

//Induction Heater Controller : E3508 

r1 := sv_IH * 10;
Tx_IH_TSV := REAL_TO_WORD(r1);

IF s_cm_RST AND is_IH_TIC_al THEN
	Tx_IH_AL_CR := 1;	
ELSE
	Tx_IH_AL_CR := 0;
END_IF

Tx_IH_ABS_HI := 1500;

END_PROGRAM

// ---- POUs/MR_PRG/P53_DO_VV.TcPOU
PROGRAM P53_DO_VV
VAR  
	p_V05, p_V06: R_TRIG;
	p_V08, p_V09: R_TRIG;
	p_V11, p_V12: R_TRIG;
	p_V14, p_V15: R_TRIG;
	p_V17, p_V18: R_TRIG;
	p_V20, p_V21: R_TRIG;
	
	n_V05, n_V06: F_TRIG;
	n_V08, n_V09: F_TRIG;
	n_V11, n_V12: F_TRIG;
	n_V14, n_V15: F_TRIG;
	n_V17, n_V18: F_TRIG;
	n_V20, n_V21: F_TRIG;
END_VAR

p_V05(CLK:= cm_V05); p_V06(CLK:= cm_V06);
p_V08(CLK:= cm_V08); p_V09(CLK:= cm_V09);
p_V11(CLK:= cm_V11); p_V12(CLK:= cm_V12);
p_V14(CLK:= cm_V14); p_V15(CLK:= cm_V15);
p_V17(CLK:= cm_V17); p_V18(CLK:= cm_V18);
p_V20(CLK:= cm_V20); p_V21(CLK:= cm_V21);

n_V05(CLK:= cm_V05); n_V06(CLK:= cm_V06);
n_V08(CLK:= cm_V08); n_V09(CLK:= cm_V09);
n_V11(CLK:= cm_V11); n_V12(CLK:= cm_V12);
n_V14(CLK:= cm_V14); n_V15(CLK:= cm_V15);
n_V17(CLK:= cm_V17); n_V18(CLK:= cm_V18);
n_V20(CLK:= cm_V20); n_V21(CLK:= cm_V21);

IF ing_MAINT = 0 THEN
	
	//interLock Valve Check
	IF p_V05.Q THEN cm_V06 := 1; END_IF  //V05 Open -> V06 Close
	IF n_V05.Q THEN cm_V06 := 0; END_IF	
	IF p_V06.Q THEN cm_V05 := 1; END_IF  //V06 Close -> V05 Open
	IF n_V06.Q THEN cm_V05 := 0; END_IF
		
	IF p_V08.Q THEN cm_V09 := 1; END_IF  //V08 Open -> V09 Close
	IF n_V08.Q THEN cm_V09 := 0; END_IF
	IF p_V09.Q THEN cm_V08 := 1; END_IF  //V09 Close -> V08 Open
	IF n_V09.Q THEN cm_V08 := 0; END_IF
	
	IF p_V11.Q THEN cm_V12 := 1; END_IF  //V11 Open -> V12 Close
	IF n_V11.Q THEN cm_V12 := 0; END_IF
	IF p_V12.Q THEN cm_V11 := 1; END_IF  //V12 Close -> V11 Open
	IF n_V12.Q THEN cm_V11 := 0; END_IF
	
	IF p_V14.Q THEN cm_V15 := 1; END_IF  //V14 Open -> V15 Close
	IF n_V14.Q THEN cm_V15 := 0; END_IF
	IF p_V15.Q THEN cm_V14 := 1; END_IF  //V15 Close -> V14 Open
	IF n_V15.Q THEN cm_V14 := 0; END_IF
	
	IF p_V17.Q THEN cm_V18 := 1; END_IF  //V17 Open -> V18 Close
	IF n_V17.Q THEN cm_V18 := 0; END_IF
	IF p_V18.Q THEN cm_V17 := 1; END_IF  //V18 Close -> V17 Open
	IF n_V18.Q THEN cm_V17 := 0; END_IF
	
	IF p_V20.Q THEN cm_V21 := 1; END_IF  //V20 Open -> V21 Close
	IF n_V20.Q THEN cm_V21 := 0; END_IF
	IF p_V21.Q THEN cm_V20 := 1; END_IF  //V21 Close -> V20 Open
	IF n_V21.Q THEN cm_V20 := 0; END_IF
	
	// Leak Check Valves Off
	cm_V36 := cm_V37 := cm_V38 := cm_V39 := 0;
	cm_V40 := cm_V41 := cm_V42 := cm_V43 := cm_V44 := cm_V45 := 0;
	cm_V46 := cm_V47 := cm_V48 := cm_V49 := cm_V50 := cm_V51 := cm_V52 := 0;
	 
	//Gas Safety Interlock-kjk - Danger Gas Supply Close
	IF is_DOR_VAC_ok = 0 THEN
		IF do_V01 THEN cm_V01 := 0; END_IF//H2 Supply
		IF do_V02 THEN cm_V02 := 0; END_IF//N2 Supply
		IF do_V03 THEN cm_V03 := 0; END_IF//SiH4 Supply
		IF do_V04 THEN cm_V04 := 0; END_IF//NH3 Supply	
	END_IF
 	 
END_IF

do_V01 := cm_V01;
do_V02 := cm_V02;
do_V03 := cm_V03;
do_V04 := cm_V04;
do_V05 := cm_V05;
do_V06 := cm_V06;
do_V07 := cm_V07;
do_V08 := cm_V08;
do_V09 := cm_V09;
do_V10 := cm_V10;
do_V11 := cm_V11;
do_V12 := cm_V12;
do_V13 := cm_V13;
do_V14 := cm_V14;
do_V15 := cm_V15;
do_V16 := cm_V16;
do_V17 := cm_V17;
do_V18 := cm_V18;
do_V19 := cm_V19;
do_V20 := cm_V20;
do_V21 := cm_V21;
do_V22 := cm_V22;
do_V23 := cm_V23;
do_V24 := cm_V24;
do_V25 := cm_V25;
do_V26 := cm_V26;
do_V27 := cm_V27;
do_V28 := cm_V28;
do_V29 := cm_V29;
do_V30 := cm_V30;
do_V31 := cm_V31;
do_V32 := cm_V32;
do_V33_1 := cm_V33_1;
do_V33_2 := cm_V33_2;
IF di_VP_busy = 0 THEN
	cm_V34 := 0; //DOR VAC Valve
END_IF
do_V34 := cm_V34;
do_V35 := cm_V35;
do_V36 := cm_V36;
do_V37 := cm_V37;
do_V38 := cm_V38;
do_V39 := cm_V39;
do_V40 := cm_V40;
do_V41 := cm_V41;
do_V42 := cm_V42;
do_V43 := cm_V43;
do_V44 := cm_V44;
do_V45 := cm_V45;
do_V46 := cm_V46;
do_V47 := cm_V47;
do_V48 := cm_V48;
do_V49 := cm_V49;
do_V50 := cm_V50;
do_V51 := cm_V51;
do_V52 := cm_V52;

//Solenoid block1
Tx_SOL1 := CSETBIT32(inVal32:= Tx_SOL1, bitNo:= N_SOL1[0], bitVal:= do_V01);
Tx_SOL1 := CSETBIT32(inVal32:= Tx_SOL1, bitNo:= N_SOL1[1], bitVal:= do_V02);
Tx_SOL1 := CSETBIT32(inVal32:= Tx_SOL1, bitNo:= N_SOL1[2], bitVal:= do_V03);
Tx_SOL1 := CSETBIT32(inVal32:= Tx_SOL1, bitNo:= N_SOL1[3], bitVal:= do_V04);
Tx_SOL1 := CSETBIT32(inVal32:= Tx_SOL1, bitNo:= N_SOL1[4], bitVal:= do_V05);
Tx_SOL1 := CSETBIT32(inVal32:= Tx_SOL1, bitNo:= N_SOL1[5], bitVal:= do_V06);
Tx_SOL1 := CSETBIT32(inVal32:= Tx_SOL1, bitNo:= N_SOL1[6], bitVal:= do_V07);
Tx_SOL1 := CSETBIT32(inVal32:= Tx_SOL1, bitNo:= N_SOL1[7], bitVal:= do_V08);
Tx_SOL1 := CSETBIT32(inVal32:= Tx_SOL1, bitNo:= N_SOL1[8], bitVal:= do_V09);
Tx_SOL1 := CSETBIT32(inVal32:= Tx_SOL1, bitNo:= N_SOL1[9], bitVal:= do_V10);

Tx_SOL1 := CSETBIT32(inVal32:= Tx_SOL1, bitNo:= N_SOL1[10], bitVal:= do_V11);
Tx_SOL1 := CSETBIT32(inVal32:= Tx_SOL1, bitNo:= N_SOL1[11], bitVal:= do_V12);
Tx_SOL1 := CSETBIT32(inVal32:= Tx_SOL1, bitNo:= N_SOL1[12], bitVal:= do_V13);
Tx_SOL1 := CSETBIT32(inVal32:= Tx_SOL1, bitNo:= N_SOL1[13], bitVal:= do_V14);
Tx_SOL1 := CSETBIT32(inVal32:= Tx_SOL1, bitNo:= N_SOL1[14], bitVal:= do_V15);
Tx_SOL1 := CSETBIT32(inVal32:= Tx_SOL1, bitNo:= N_SOL1[15], bitVal:= do_V16);
Tx_SOL1 := CSETBIT32(inVal32:= Tx_SOL1, bitNo:= N_SOL1[16], bitVal:= do_V36);
Tx_SOL1 := CSETBIT32(inVal32:= Tx_SOL1, bitNo:= N_SOL1[17], bitVal:= do_V37);
Tx_SOL1 := CSETBIT32(inVal32:= Tx_SOL1, bitNo:= N_SOL1[18], bitVal:= do_V38);
Tx_SOL1 := CSETBIT32(inVal32:= Tx_SOL1, bitNo:= N_SOL1[19], bitVal:= do_V39);

Tx_SOL1 := CSETBIT32(inVal32:= Tx_SOL1, bitNo:= N_SOL1[20], bitVal:= do_V40);
Tx_SOL1 := CSETBIT32(inVal32:= Tx_SOL1, bitNo:= N_SOL1[21], bitVal:= do_V41);
Tx_SOL1 := CSETBIT32(inVal32:= Tx_SOL1, bitNo:= N_SOL1[22], bitVal:= do_V42);
Tx_SOL1 := CSETBIT32(inVal32:= Tx_SOL1, bitNo:= N_SOL1[23], bitVal:= do_V43);
Tx_SOL1 := CSETBIT32(inVal32:= Tx_SOL1, bitNo:= N_SOL1[24], bitVal:= do_V44);
Tx_SOL1 := CSETBIT32(inVal32:= Tx_SOL1, bitNo:= N_SOL1[25], bitVal:= do_V45);

//Solenoid block2
Tx_SOL2 := CSETBIT32(inVal32:= Tx_SOL2, bitNo:= N_SOL2[0], bitVal:= do_V17);
Tx_SOL2 := CSETBIT32(inVal32:= Tx_SOL2, bitNo:= N_SOL2[1], bitVal:= do_V18);
Tx_SOL2 := CSETBIT32(inVal32:= Tx_SOL2, bitNo:= N_SOL2[2], bitVal:= do_V19);
Tx_SOL2 := CSETBIT32(inVal32:= Tx_SOL2, bitNo:= N_SOL2[3], bitVal:= do_V20);
Tx_SOL2 := CSETBIT32(inVal32:= Tx_SOL2, bitNo:= N_SOL2[4], bitVal:= do_V21);
Tx_SOL2 := CSETBIT32(inVal32:= Tx_SOL2, bitNo:= N_SOL2[5], bitVal:= do_V22);
Tx_SOL2 := CSETBIT32(inVal32:= Tx_SOL2, bitNo:= N_SOL2[6], bitVal:= do_V23);
Tx_SOL2 := CSETBIT32(inVal32:= Tx_SOL2, bitNo:= N_SOL2[7], bitVal:= do_V24);
Tx_SOL2 := CSETBIT32(inVal32:= Tx_SOL2, bitNo:= N_SOL2[8], bitVal:= do_V25);
Tx_SOL2 := CSETBIT32(inVal32:= Tx_SOL2, bitNo:= N_SOL2[9], bitVal:= do_V26);

Tx_SOL2 := CSETBIT32(inVal32:= Tx_SOL2, bitNo:= N_SOL2[10], bitVal:= do_V27);
Tx_SOL2 := CSETBIT32(inVal32:= Tx_SOL2, bitNo:= N_SOL2[11], bitVal:= do_V28);
Tx_SOL2 := CSETBIT32(inVal32:= Tx_SOL2, bitNo:= N_SOL2[12], bitVal:= do_V29);
Tx_SOL2 := CSETBIT32(inVal32:= Tx_SOL2, bitNo:= N_SOL2[13], bitVal:= do_V30);
Tx_SOL2 := CSETBIT32(inVal32:= Tx_SOL2, bitNo:= N_SOL2[14], bitVal:= do_V31);
Tx_SOL2 := CSETBIT32(inVal32:= Tx_SOL2, bitNo:= N_SOL2[15], bitVal:= do_V32);
Tx_SOL2 := CSETBIT32(inVal32:= Tx_SOL2, bitNo:= N_SOL2[16], bitVal:= do_V33_1);
Tx_SOL2 := CSETBIT32(inVal32:= Tx_SOL2, bitNo:= N_SOL2[17], bitVal:= do_V33_2);
Tx_SOL2 := CSETBIT32(inVal32:= Tx_SOL2, bitNo:= N_SOL2[18], bitVal:= do_V34);
Tx_SOL2 := CSETBIT32(inVal32:= Tx_SOL2, bitNo:= N_SOL2[19], bitVal:= do_V35);

Tx_SOL2 := CSETBIT32(inVal32:= Tx_SOL2, bitNo:= N_SOL2[20], bitVal:= do_V46);
Tx_SOL2 := CSETBIT32(inVal32:= Tx_SOL2, bitNo:= N_SOL2[21], bitVal:= do_V47);
Tx_SOL2 := CSETBIT32(inVal32:= Tx_SOL2, bitNo:= N_SOL2[22], bitVal:= do_V48);
Tx_SOL2 := CSETBIT32(inVal32:= Tx_SOL2, bitNo:= N_SOL2[23], bitVal:= do_V49);
Tx_SOL2 := CSETBIT32(inVal32:= Tx_SOL2, bitNo:= N_SOL2[24], bitVal:= do_V50);
Tx_SOL2 := CSETBIT32(inVal32:= Tx_SOL2, bitNo:= N_SOL2[25], bitVal:= do_V51);
Tx_SOL2 := CSETBIT32(inVal32:= Tx_SOL2, bitNo:= N_SOL2[26], bitVal:= do_V52);

END_PROGRAM

// ---- POUs/MR_PRG/P54_DO_ETC.TcPOU
PROGRAM P54_DO_ETC
VAR
	is_ROT_ON: BOOL;
	
	p_RC_lamp: R_TRIG; //by Button
	p_GC_lamp: R_TRIG; //by Button
	on_RC_lamp: BOOL; //by Button
	on_GC_lamp: BOOL; //by Button
	
	//For Blue Signal & Reset Lamp
	T_BU_on: TON := (PT:= T#1S);
	T_BU_off: TON := (PT:= T#1S);
END_VAR

p_RC_lamp(CLK:= di_RC_lamp);
p_GC_lamp(CLK:= di_GC_lamp);

IF p_RC_lamp.Q THEN
	on_RC_lamp := NOT on_RC_lamp;
END_IF

IF p_GC_lamp.Q THEN
	on_GC_lamp := NOT on_GC_lamp;
END_IF


IF ing_Maint THEN	 
	 IF s_EN_DO_TEST THEN // MaintMode -> D/O PC TEST 
	  	is_ROT_ON := cm_ROT OR s_EN_ROT_JOG OR s_EN_ROT_INCH OR s_EN_EXE_ROT_CALI;// AND b_ALARM_ON; //test
	 ELSE
	  	cm_RED := cm_YE := cm_GN := cm_BU := cm_WH := cm_BZ := 0;
		is_ROT_ON := cm_ROT OR s_EN_ROT_JOG OR s_EN_ROT_INCH OR s_EN_EXE_ROT_CALI;// AND b_ALARM_ON; //test
	 END_IF  	 
ELSE
	 cm_RED := is_AL;
	 cm_YE := is_WN;
	 cm_GN := ing_RCP;
	 //cm_BU := ing_MAINT;	 
	 //cm_BZ := p_NewAL_Risec -> Cause_N_Effect에서 처리
	 //END_IF
	 //IF cm_BZ_OFF THEN
	 // cm_BZ := Off;
	  //cm_BZ_OFF := Off; 
	 //END_IF

 	//cm_IHT_ON := b_AL = 0; -> Cause_N_Effect에서 처리    
 	is_ROT_ON := cm_ROT OR s_EN_ROT_JOG OR s_EN_ROT_INCH OR s_EN_EXE_ROT_CALI;// AND b_ALARM_ON; //test
END_IF

cm_WH := ing_MAINT;

T_BU_on(IN:= (is_AL OR is_WN) AND T_BU_off.Q = 0);
T_BU_off(IN:= T_BU_on.Q);

do_RED := cm_RED;
do_YE := cm_YE;//------------------------------------
do_GN := cm_GN;
do_BU := cm_BU OR ((is_AL OR is_WN) AND T_BU_on.Q = 0);//------------------------------------
do_WH := cm_WH;//------------------------------------
do_BZ := cm_BZ;

do_SH_up_ry := cm_SH_up_ry;//------------------------------------
do_SH_dw_ry := cm_SH_dw_ry;//------------------------------------

do_IH := cm_IH;
do_IH_rst := cm_IH_rst OR (di_IH_fail AND s_cm_RST);

do_VP := cm_VP;
do_VP_rst := cm_VP_rst OR ((di_VP_fail = 1 OR di_VP_al = 0 OR di_VP_wn = 0) AND s_cm_RST);//------------------------------------

do_SYS_off_lock := cm_SYS_off_lock OR ing_RCP;//----------------------------------------

do_RC_lamp := cm_RC_lamp OR on_RC_lamp OR (e_d_AUTO_RC_LAMP_on AND di_RC_close = 0) ;//----------------------------------------
do_GC_lamp := cm_GC_lamp OR on_GC_lamp OR (e_d_AUTO_GC_LAMP_on AND di_GC_close = 0);//----------------------------------------
do_CC_lamp := cm_CC_lamp OR di_CC_close = 0;//----------------------------------------

do_IH_mc := cm_IH_mc;//----------------------------------------
do_TB_mc := cm_TB_mc;//----------------------------------------
do_VP_mc := cm_VP_mc;//----------------------------------------
do_LH_mc := cm_LH_mc;//----------------------------------------

do_ROT := cm_ROT OR is_ROT_ON;// -> 위에서 처리 
do_ROT_break := do_ROT;//cm_ROT_break;//----------------------------------------
do_ROT_rst := cm_ROT_rst OR (di_ROT_fail = 0 AND s_cm_RST);//----------------------------------------

do_RST_led := cm_RST_led OR di_RST OR ((is_AL OR is_WN) AND T_BU_on.Q = 0);//----------------------------------------
do_DOR_VAC_led := cm_DOR_VAC_led OR (s_EN_EXE_DOR_VAC AND is_DOR_VAC_blink) OR (s_EN_EXE_DOR_VAC = 0 AND is_DOR_05ATM);//----------------------------------------
do_DOR_ATM_led := cm_DOR_ATM_led OR (s_EN_EXE_DOR_ATM AND is_DOR_ATM_blink) OR (s_EN_EXE_DOR_ATM = 0 AND is_DOR_1ATM);//----------------------------------------

do_SH_up_led := cm_SH_up_led;//----------------------------------------
do_SH_dw_led := cm_SH_dw_led;//----------------------------------------

//Real Output*******************
%QB0 := BITS1_DO;
%QB1 := BITS2_DO;
%QB2 := BITS3_DO;
%QB3 := BITS4_DO;

END_PROGRAM

// ---- POUs/MR_PRG/P61_AO.TcPOU
PROGRAM P61_AO
VAR
	//ACT_Ramp_OLD();
	MFC01, MFC02, MFC03, MFC04, MFC05, MFC06, MFC07, MFC08, MFC09, MFC10: FB_Ramp2;
	MFC11, MFC12, MFC13, MFC14, MFC15, MFC16, MFC17, MFC18, MFC19: FB_Ramp2;		
	EPC01, EPC02, EPC03, EPC04, EPC05, EPC06, EPC07: FB_Ramp2;	
	IH, ROT, POS, P01: FB_Ramp2;
		
	//HT01: FB_Ramp2;
	halfRes: REAL := 16383;//0~5V
	fullRes: REAL := 32767;//0~10V or 4~20mA
	halfRes_ROT: REAL := 13106;//0~4V : 0 ~ 2500RPM - BLHM230K-GFS
		
	M01, M02, M03, M04, M05, M06, M07, M08, M09, M10: FB_Ramp_0;
	M11, M12, M13, M14, M15, M16, M17, M18, M19: FB_Ramp_0;	
	E01, E02, E03, E04, E05, E06, E07: FB_Ramp_0;	
	IH_0, ROT_0, POS_0, P01_0: FB_Ramp_0;
END_VAR

//IF EN_RUN_RCP = Off THEN
	ACT_Ramp();
//	ACT_Ramp_OLD();	
//END_IF

//----------------------------Analog Output--------------------------
IF N_MAX[0] > 0 THEN YA_M01 := REAL_TO_WORD(sv_M01 * halfRes / N_MAX[0]); END_IF;//MFC01 : 0~5V
IF N_MAX[1] > 0 THEN YA_M02 := REAL_TO_WORD(sv_M02 * halfRes / N_MAX[1]); END_IF;//MFC02 : 0~5V
IF N_MAX[2] > 0 THEN YA_M03 := REAL_TO_WORD(sv_M03 * halfRes / N_MAX[2]); END_IF;//MFC03 : 0~5V
IF N_MAX[3] > 0 THEN YA_M04 := REAL_TO_WORD(sv_M04 * halfRes / N_MAX[3]); END_IF;//MFC04 : 0~5V
IF N_MAX[4] > 0 THEN YA_M05 := REAL_TO_WORD(sv_M05 * halfRes / N_MAX[4]); END_IF;//MFC05 : 0~5V
IF N_MAX[5] > 0 THEN YA_M06 := REAL_TO_WORD(sv_M06 * halfRes / N_MAX[5]); END_IF;//MFC06 : 0~5V
IF N_MAX[6] > 0 THEN YA_M07 := REAL_TO_WORD(sv_M07 * halfRes / N_MAX[6]); END_IF;//MFC07 : 0~5V       
IF N_MAX[7] > 0 THEN YA_M08 := REAL_TO_WORD(sv_M08 * halfRes / N_MAX[7]); END_IF;//MFC08 : 0~5V
IF N_MAX[8] > 0 THEN YA_M09 := REAL_TO_WORD(sv_M09 * halfRes / N_MAX[8]); END_IF;//MFC09 : 0~5V
IF N_MAX[9] > 0 THEN YA_M10 := REAL_TO_WORD(sv_M10 * halfRes / N_MAX[9]); END_IF;//MFC10 : 0~5V
IF N_MAX[10] > 0 THEN YA_M11 := REAL_TO_WORD(sv_M11 * halfRes / N_MAX[10]); END_IF;//MFC11 : 0~5V
IF N_MAX[11] > 0 THEN YA_M12 := REAL_TO_WORD(sv_M12 * halfRes / N_MAX[11]); END_IF;//MFC12 : 0~5V
IF N_MAX[12] > 0 THEN YA_M13 := REAL_TO_WORD(sv_M13 * halfRes / N_MAX[12]); END_IF;//MFC13 : 0~5V
IF N_MAX[13] > 0 THEN YA_M14 := REAL_TO_WORD(sv_M14 * halfRes / N_MAX[13]); END_IF;//MFC14 : 0~5V
IF N_MAX[14] > 0 THEN YA_M15 := REAL_TO_WORD(sv_M15 * halfRes / N_MAX[14]); END_IF;//MFC15 : 0~5V
IF N_MAX[15] > 0 THEN YA_M16 := REAL_TO_WORD(sv_M16 * halfRes / N_MAX[15]); END_IF;//MFC16 : 0~5V
IF N_MAX[16] > 0 THEN YA_M17 := REAL_TO_WORD(sv_M17 * halfRes / N_MAX[16]); END_IF;//MFC17 : 0~5V
IF N_MAX[17] > 0 THEN YA_M18 := REAL_TO_WORD(sv_M18 * halfRes / N_MAX[17]); END_IF;//MFC18 : 0~5V
IF N_MAX[18] > 0 THEN YA_M19 := REAL_TO_WORD(sv_M19 * halfRes / N_MAX[18]); END_IF;//MFC19 : 0~5V
IF N_MAX[19] > 0 THEN YA_E01 := REAL_TO_WORD(sv_E01 * halfRes / N_MAX[19]); END_IF;//EPC01 : 0~5V
IF N_MAX[20] > 0 THEN YA_E02 := REAL_TO_WORD(sv_E02 * halfRes / N_MAX[20]); END_IF;//EPC02 : 0~5V
IF N_MAX[21] > 0 THEN YA_E03 := REAL_TO_WORD(sv_E03 * halfRes / N_MAX[21]); END_IF;//EPC03 : 0~5V
IF N_MAX[22] > 0 THEN YA_E04 := REAL_TO_WORD(sv_E04 * halfRes / N_MAX[22]); END_IF;//EPC04 : 0~5V
IF N_MAX[23] > 0 THEN YA_E05 := REAL_TO_WORD(sv_E05 * halfRes / N_MAX[23]); END_IF;//EPC05 : 0~5V
IF N_MAX[24] > 0 THEN YA_E06 := REAL_TO_WORD(sv_E06 * halfRes / N_MAX[24]); END_IF;//EPC06 : 0~5V
IF N_MAX[25] > 0 THEN YA_E07 := REAL_TO_WORD(sv_E07 * halfRes / N_MAX[25]); END_IF;//EPC07 : 0~5V
YA_P03 := XA_P03;//Exhaust Pressure(1000 Torr) Display-> AM215A-13  : 0~10V  
//IF N_MAX[26] > 0 THEN YA_Temp := REAL_TO_WORD(sv_IHT * fullRes / N_MAX[26]); END_IF;//IH - E3508 - DeviceNet
IF N_MAX[27] > 0 THEN YA_ROT := REAL_TO_WORD(e_ROT_AO_OFFSET + (sv_ROT * halfRes_ROT / N_MAX[27]) * e_ROT_AO_SLOPE_FACTOR); END_IF;//ROT : 0~4V
//IF N_MAX[27] > 0 THEN YA_ROT := REAL_TO_WORD(sv_ROT * halfRes_ROT / N_MAX[27]); END_IF;//ROT : 0~4V
//IF N_MAX[28] > 0 THEN YA_TV := REAL_TO_WORD(sv_TV * fullRes / N_MAX[28]); END_IF;//TV Position- Nocal - DeviceNet
//IF N_MAX[29] > 0 THEN YA_P01 := REAL_TO_WORD(sv_P01 * fullRes / N_MAX[29]); END_IF;//TV Pressure- Nocal - DeviceNet

ACTION ACT_Ramp:
